   1:L PR[91] R[100]mm/sec CNT100;
   1:  PR[91,1] = PR[90,1] + 58.118;
   1:  PR[91,2] = PR[90,2] + -22.323;
   1:  PR[91,3] = PR[90,3] + 45.021;
   1:L PR[91] R[100]mm/sec CNT100;
   1:  PR[91,1] = PR[90,1] + 59.291;
   1:  PR[91,2] = PR[90,2] + -22.455;
   1:  PR[91,3] = PR[90,3] + 45.028;
   1:L PR[91] R[100]mm/sec CNT100;
   1:  PR[91,1] = PR[90,1] + 63.095;
   1:  PR[91,2] = PR[90,2] + -22.522;
   1:  PR[91,3] = PR[90,3] + 45.032;
   1:L PR[91] R[100]mm/sec CNT100;
   1:  PR[91,1] = PR[90,1] + 66.999;
   1:  PR[91,2] = PR[90,2] + -22.167;
   1:  PR[91,3] = PR[90,3] + 45.043;
   1:L PR[91] R[100]mm/sec CNT100;
   1:  PR[91,1] = PR[90,1] + 68.277;
   1:  PR[91,2] = PR[90,2] + -21.945;
   1:  PR[91,3] = PR[90,3] + 45.054;
   1:L PR[91] R[100]mm/sec CNT100;
   1:  PR[91,1] = PR[90,1] + 73.428;
   1:  PR[91,2] = PR[90,2] + -20.409;
   1:  PR[91,3] = PR[90,3] + 45.058;
   1:L PR[91] R[100]mm/sec CNT100;
   1:  PR[91,1] = PR[90,1] + 73.641;
   1:  PR[91,2] = PR[90,2] + -20.327;
   1:  PR[91,3] = PR[90,3] + 45.073;
   1:L PR[91] R[100]mm/sec CNT100;
   1:  PR[91,1] = PR[90,1] + 77.548;
   1:  PR[91,2] = PR[90,2] + -18.168;
   1:  PR[91,3] = PR[90,3] + 45.074;
   1:L PR[91] R[100]mm/sec CNT100;
   1:  PR[91,1] = PR[90,1] + 78.651;
   1:  PR[91,2] = PR[90,2] + -17.462;
   1:  PR[91,3] = PR[90,3] + 45.087;
   1:L PR[91] R[100]mm/sec CNT100;
   1:  PR[91,1] = PR[90,1] + 81.067;
   1:  PR[91,2] = PR[90,2] + -15.304;
   1:  PR[91,3] = PR[90,3] + 45.091;
   1:L PR[91] R[100]mm/sec CNT100;
   1:  PR[91,1] = PR[90,1] + 82.534;
   1:  PR[91,2] = PR[90,2] + -13.852;
   1:  PR[91,3] = PR[90,3] + 45.100;
   1:L PR[91] R[100]mm/sec CNT100;
   1:  PR[91,1] = PR[90,1] + 83.900;
   1:  PR[91,2] = PR[90,2] + -11.894;
   1:  PR[91,3] = PR[90,3] + 45.106;
   1:L PR[91] R[100]mm/sec CNT100;
   1:  PR[91,1] = PR[90,1] + 85.291;
   1:  PR[91,2] = PR[90,2] + -9.736;
   1:  PR[91,3] = PR[90,3] + 45.113;
   1:L PR[91] R[100]mm/sec CNT100;
   1:  PR[91,1] = PR[90,1] + 85.955;
   1:  PR[91,2] = PR[90,2] + -8.019;
   1:  PR[91,3] = PR[90,3] + 45.121;
   1:L PR[91] R[100]mm/sec CNT100;
   1:  PR[91,1] = PR[90,1] + 86.933;
   1:  PR[91,2] = PR[90,2] + -5.315;
   1:  PR[91,3] = PR[90,3] + 45.126;
   1:L PR[91] R[100]mm/sec CNT100;
   1:  PR[91,1] = PR[90,1] + 87.308;
   1:  PR[91,2] = PR[90,2] + -2.135;
   1:  PR[91,3] = PR[90,3] + 45.134;
   1:L PR[91] R[100]mm/sec CNT100;
   1:  PR[91,1] = PR[90,1] + 87.416;
   1:  PR[91,2] = PR[90,2] + -1.644;
   1:  PR[91,3] = PR[90,3] + 45.144;
   1:L PR[91] R[100]mm/sec CNT100;
   1:  PR[91,1] = PR[90,1] + 87.528;
   1:  PR[91,2] = PR[90,2] + -0.738;
   1:  PR[91,3] = PR[90,3] + 45.145;
   1:L PR[91] R[100]mm/sec CNT100;
   1:  PR[91,1] = PR[90,1] + 87.126;
   1:  PR[91,2] = PR[90,2] + 2.303;
   1:  PR[91,3] = PR[90,3] + 45.148;
   1:L PR[91] R[100]mm/sec CNT100;
   1:  PR[91,1] = PR[90,1] + 86.935;
   1:  PR[91,2] = PR[90,2] + 3.851;
   1:  PR[91,3] = PR[90,3] + 45.157;
   1:L PR[91] R[100]mm/sec CNT100;
   1:  PR[91,1] = PR[90,1] + 85.955;
   1:  PR[91,2] = PR[90,2] + 6.560;
   1:  PR[91,3] = PR[90,3] + 45.161;
   1:L PR[91] R[100]mm/sec CNT100;
   1:  PR[91,1] = PR[90,1] + 85.291;
   1:  PR[91,2] = PR[90,2] + 8.277;
   1:  PR[91,3] = PR[90,3] + 45.169;
   1:L PR[91] R[100]mm/sec CNT100;
   1:  PR[91,1] = PR[90,1] + 83.900;
   1:  PR[91,2] = PR[90,2] + 10.435;
   1:  PR[91,3] = PR[90,3] + 45.175;
   1:L PR[91] R[100]mm/sec CNT100;
   1:  PR[91,1] = PR[90,1] + 82.534;
   1:  PR[91,2] = PR[90,2] + 12.393;
   1:  PR[91,3] = PR[90,3] + 45.182;
   1:L PR[91] R[100]mm/sec CNT100;
   1:  PR[91,1] = PR[90,1] + 81.067;
   1:  PR[91,2] = PR[90,2] + 13.845;
   1:  PR[91,3] = PR[90,3] + 45.189;
   1:L PR[91] R[100]mm/sec CNT100;
   1:  PR[91,1] = PR[90,1] + 78.651;
   1:  PR[91,2] = PR[90,2] + 16.003;
   1:  PR[91,3] = PR[90,3] + 45.195;
   1:L PR[91] R[100]mm/sec CNT100;
   1:  PR[91,1] = PR[90,1] + 77.549;
   1:  PR[91,2] = PR[90,2] + 16.709;
   1:  PR[91,3] = PR[90,3] + 45.205;
   1:L PR[91] R[100]mm/sec CNT100;
   1:  PR[91,1] = PR[90,1] + 73.642;
   1:  PR[91,2] = PR[90,2] + 18.868;
   1:  PR[91,3] = PR[90,3] + 45.208;
   1:L PR[91] R[100]mm/sec CNT100;
   1:  PR[91,1] = PR[90,1] + 73.428;
   1:  PR[91,2] = PR[90,2] + 18.950;
   1:  PR[91,3] = PR[90,3] + 45.221;
   1:L PR[91] R[100]mm/sec CNT100;
   1:  PR[91,1] = PR[90,1] + 68.270;
   1:  PR[91,2] = PR[90,2] + 20.489;
   1:  PR[91,3] = PR[90,3] + 45.222;
   1:L PR[91] R[100]mm/sec CNT100;
   1:  PR[91,1] = PR[90,1] + 66.977;
   1:  PR[91,2] = PR[90,2] + 20.710;
   1:  PR[91,3] = PR[90,3] + 45.238;
   1:L PR[91] R[100]mm/sec CNT100;
   1:  PR[91,1] = PR[90,1] + 63.068;
   1:  PR[91,2] = PR[90,2] + 21.066;
   1:  PR[91,3] = PR[90,3] + 45.241;
   1:L PR[91] R[100]mm/sec CNT100;
   1:  PR[91,1] = PR[90,1] + 59.214;
   1:  PR[91,2] = PR[90,2] + 20.989;
   1:  PR[91,3] = PR[90,3] + 45.253;
   1:L PR[91] R[100]mm/sec CNT100;
   1:  PR[91,1] = PR[90,1] + 58.065;
   1:  PR[91,2] = PR[90,2] + 20.860;
   1:  PR[91,3] = PR[90,3] + 45.264;
   1:L PR[91] R[100]mm/sec CNT100;
   1:  PR[91,1] = PR[90,1] + 55.759;
   1:  PR[91,2] = PR[90,2] + 20.363;
   1:  PR[91,3] = PR[90,3] + 45.267;
   1:L PR[91] R[100]mm/sec CNT100;
   1:  PR[91,1] = PR[90,1] + 53.207;
   1:  PR[91,2] = PR[90,2] + 19.893;
   1:  PR[91,3] = PR[90,3] + 45.274;
   1:L PR[91] R[100]mm/sec CNT100;
   1:  PR[91,1] = PR[90,1] + 51.984;
   1:  PR[91,2] = PR[90,2] + 19.647;
   1:  PR[91,3] = PR[90,3] + 45.282;
   1:L PR[91] R[100]mm/sec CNT100;
   1:  PR[91,1] = PR[90,1] + 49.065;
   1:  PR[91,2] = PR[90,2] + 18.507;
   1:  PR[91,3] = PR[90,3] + 45.285;
   1:L PR[91] R[100]mm/sec CNT100;
   1:  PR[91,1] = PR[90,1] + 45.352;
   1:  PR[91,2] = PR[90,2] + 16.958;
   1:  PR[91,3] = PR[90,3] + 45.294;
   1:L PR[91] R[100]mm/sec CNT100;
   1:  PR[91,1] = PR[90,1] + 44.475;
   1:  PR[91,2] = PR[90,2] + 16.351;
   1:  PR[91,3] = PR[90,3] + 45.306;
   1:L PR[91] R[100]mm/sec CNT100;
   1:  PR[91,1] = PR[90,1] + 39.433;
   1:  PR[91,2] = PR[90,2] + 13.177;
   1:  PR[91,3] = PR[90,3] + 45.309;
   1:L PR[91] R[100]mm/sec CNT100;
   1:  PR[91,1] = PR[90,1] + 37.041;
   1:  PR[91,2] = PR[90,2] + 15.548;
   1:  PR[91,3] = PR[90,3] + 45.327;
   1:L PR[91] R[100]mm/sec CNT100;
   1:  PR[91,1] = PR[90,1] + 35.593;
   1:  PR[91,2] = PR[90,2] + 16.643;
   1:  PR[91,3] = PR[90,3] + 45.336;
   1:L PR[91] R[100]mm/sec CNT100;
   1:  PR[91,1] = PR[90,1] + 34.665;
   1:  PR[91,2] = PR[90,2] + 17.312;
   1:  PR[91,3] = PR[90,3] + 45.342;
   1:L PR[91] R[100]mm/sec CNT100;
   1:  PR[91,1] = PR[90,1] + 34.298;
   1:  PR[91,2] = PR[90,2] + 17.553;
   1:  PR[91,3] = PR[90,3] + 45.345;
   1:L PR[91] R[100]mm/sec CNT100;
   1:  PR[91,1] = PR[90,1] + 31.694;
   1:  PR[91,2] = PR[90,2] + 18.777;
   1:  PR[91,3] = PR[90,3] + 45.346;
   1:L PR[91] R[100]mm/sec CNT100;
   1:  PR[91,1] = PR[90,1] + 29.317;
   1:  PR[91,2] = PR[90,2] + 19.751;
   1:  PR[91,3] = PR[90,3] + 45.355;
   1:L PR[91] R[100]mm/sec CNT100;
   1:  PR[91,1] = PR[90,1] + 26.382;
   1:  PR[91,2] = PR[90,2] + 20.320;
   1:  PR[91,3] = PR[90,3] + 45.362;
   1:L PR[91] R[100]mm/sec CNT100;
   1:  PR[91,1] = PR[90,1] + 24.007;
   1:  PR[91,2] = PR[90,2] + 20.632;
   1:  PR[91,3] = PR[90,3] + 45.371;
   1:L PR[91] R[100]mm/sec CNT100;
   1:  PR[91,1] = PR[90,1] + 20.837;
   1:  PR[91,2] = PR[90,2] + 20.451;
   1:  PR[91,3] = PR[90,3] + 45.378;
   1:L PR[91] R[100]mm/sec CNT100;
   1:  PR[91,1] = PR[90,1] + 18.643;
   1:  PR[91,2] = PR[90,2] + 20.167;
   1:  PR[91,3] = PR[90,3] + 45.387;
   1:L PR[91] R[100]mm/sec CNT100;
   1:  PR[91,1] = PR[90,1] + 15.437;
   1:  PR[91,2] = PR[90,2] + 19.153;
   1:  PR[91,3] = PR[90,3] + 45.393;
   1:L PR[91] R[100]mm/sec CNT100;
   1:  PR[91,1] = PR[90,1] + 13.560;
   1:  PR[91,2] = PR[90,2] + 18.384;
   1:  PR[91,3] = PR[90,3] + 45.403;
   1:L PR[91] R[100]mm/sec CNT100;
   1:  PR[91,1] = PR[90,1] + 10.558;
   1:  PR[91,2] = PR[90,2] + 16.515;
   1:  PR[91,3] = PR[90,3] + 45.409;
   1:L PR[91] R[100]mm/sec CNT100;
   1:  PR[91,1] = PR[90,1] + 9.078;
   1:  PR[91,2] = PR[90,2] + 15.390;
   1:  PR[91,3] = PR[90,3] + 45.419;
   1:L PR[91] R[100]mm/sec CNT100;
   1:  PR[91,1] = PR[90,1] + 6.497;
   1:  PR[91,2] = PR[90,2] + 12.675;
   1:  PR[91,3] = PR[90,3] + 45.425;
   1:L PR[91] R[100]mm/sec CNT100;
   1:  PR[91,1] = PR[90,1] + 5.421;
   1:  PR[91,2] = PR[90,2] + 11.285;
   1:  PR[91,3] = PR[90,3] + 45.435;
   1:L PR[91] R[100]mm/sec CNT100;
   1:  PR[91,1] = PR[90,1] + 5.280;
   1:  PR[91,2] = PR[90,2] + 11.075;
   1:  PR[91,3] = PR[90,3] + 45.441;
   1:L PR[91] R[100]mm/sec CNT100;
   1:  PR[91,1] = PR[90,1] + 5.067;
   1:  PR[91,2] = PR[90,2] + 10.734;
   1:L PR[91] R[100]mm/sec CNT100;
   1:  PR[91,1] = PR[90,1] + 2.658;
   1:  PR[91,2] = PR[90,2] + 6.129;
   1:  PR[91,3] = PR[90,3] + 45.442;
   1:L PR[91] R[100]mm/sec CNT100;
   1:  PR[91,1] = PR[90,1] + 0.301;
   1:  PR[91,2] = PR[90,2] + 10.494;
   1:  PR[91,3] = PR[90,3] + 45.457;
   1:L PR[91] R[100]mm/sec CNT100;
   1:  PR[91,1] = PR[90,1] + -0.405;
   1:  PR[91,2] = PR[90,2] + 11.362;
   1:  PR[91,3] = PR[90,3] + 45.472;
   1:L PR[91] R[100]mm/sec CNT100;
   1:  PR[91,1] = PR[90,1] + -2.903;
   1:  PR[91,2] = PR[90,2] + 14.051;
   1:  PR[91,3] = PR[90,3] + 45.475;
   1:L PR[91] R[100]mm/sec CNT100;
   1:  PR[91,1] = PR[90,1] + -4.419;
   1:  PR[91,2] = PR[90,2] + 15.218;
   1:  PR[91,3] = PR[90,3] + 45.486;
   1:L PR[91] R[100]mm/sec CNT100;
   1:  PR[91,1] = PR[90,1] + -6.800;
   1:  PR[91,2] = PR[90,2] + 16.795;
   1:  PR[91,3] = PR[90,3] + 45.491;
   1:L PR[91] R[100]mm/sec CNT100;
   1:  PR[91,1] = PR[90,1] + -9.296;
   1:  PR[91,2] = PR[90,2] + 17.953;
   1:  PR[91,3] = PR[90,3] + 45.500;
   1:L PR[91] R[100]mm/sec CNT100;
   1:  PR[91,1] = PR[90,1] + -11.158;
   1:  PR[91,2] = PR[90,2] + 18.656;
   1:  PR[91,3] = PR[90,3] + 45.508;
   1:L PR[91] R[100]mm/sec CNT100;
   1:  PR[91,1] = PR[90,1] + -14.668;
   1:  PR[91,2] = PR[90,2] + 19.438;
   1:  PR[91,3] = PR[90,3] + 45.513;
   1:L PR[91] R[100]mm/sec CNT100;
   1:  PR[91,1] = PR[90,1] + -15.765;
   1:  PR[91,2] = PR[90,2] + 19.597;
   1:  PR[91,3] = PR[90,3] + 45.524;
   1:L PR[91] R[100]mm/sec CNT100;
   1:  PR[91,1] = PR[90,1] + -20.138;
   1:  PR[91,2] = PR[90,2] + 19.641;
   1:  PR[91,3] = PR[90,3] + 45.527;
   1:L PR[91] R[100]mm/sec CNT100;
   1:  PR[91,1] = PR[90,1] + -20.417;
   1:  PR[91,2] = PR[90,2] + 19.622;
   1:  PR[91,3] = PR[90,3] + 45.540;
   1:L PR[91] R[100]mm/sec CNT100;
   1:  PR[91,1] = PR[90,1] + -25.039;
   1:  PR[91,2] = PR[90,2] + 18.709;
   1:  PR[91,3] = PR[90,3] + 45.541;
   1:L PR[91] R[100]mm/sec CNT100;
   1:  PR[91,1] = PR[90,1] + -29.184;
   1:  PR[91,2] = PR[90,2] + 16.938;
   1:  PR[91,3] = PR[90,3] + 45.554;
   1:L PR[91] R[100]mm/sec CNT100;
   1:  PR[91,1] = PR[90,1] + -29.594;
   1:  PR[91,2] = PR[90,2] + 16.676;
   1:  PR[91,3] = PR[90,3] + 45.567;
   1:L PR[91] R[100]mm/sec CNT100;
   1:  PR[91,1] = PR[90,1] + -32.833;
   1:  PR[91,2] = PR[90,2] + 14.369;
   1:  PR[91,3] = PR[90,3] + 45.569;
   1:L PR[91] R[100]mm/sec CNT100;
   1:  PR[91,1] = PR[90,1] + -33.458;
   1:  PR[91,2] = PR[90,2] + 13.742;
   1:  PR[91,3] = PR[90,3] + 45.580;
   1:L PR[91] R[100]mm/sec CNT100;
   1:  PR[91,1] = PR[90,1] + -35.840;
   1:  PR[91,2] = PR[90,2] + 11.109;
   1:  PR[91,3] = PR[90,3] + 45.583;
   1:L PR[91] R[100]mm/sec CNT100;
   1:  PR[91,1] = PR[90,1] + -36.555;
   1:  PR[91,2] = PR[90,2] + 9.975;
   1:  PR[91,3] = PR[90,3] + 45.593;
   1:L PR[91] R[100]mm/sec CNT100;
   1:  PR[91,1] = PR[90,1] + -36.941;
   1:  PR[91,2] = PR[90,2] + 9.506;
   1:  PR[91,3] = PR[90,3] + 45.597;
   1:L PR[91] R[100]mm/sec CNT100;
   1:  PR[91,1] = PR[90,1] + -37.589;
   1:  PR[91,2] = PR[90,2] + 8.519;
   1:  PR[91,3] = PR[90,3] + 45.599;
   1:L PR[91] R[100]mm/sec CNT100;
   1:  PR[91,1] = PR[90,1] + -38.983;
   1:  PR[91,2] = PR[90,2] + 5.816;
   1:  PR[91,3] = PR[90,3] + 45.602;
   1:L PR[91] R[100]mm/sec CNT100;
   1:  PR[91,1] = PR[90,1] + -43.442;
   1:  PR[91,2] = PR[90,2] + 11.098;
   1:  PR[91,3] = PR[90,3] + 45.611;
   1:L PR[91] R[100]mm/sec CNT100;
   1:  PR[91,1] = PR[90,1] + -43.553;
   1:  PR[91,2] = PR[90,2] + 11.183;
   1:  PR[91,3] = PR[90,3] + 45.631;
   1:L PR[91] R[100]mm/sec CNT100;
   1:  PR[91,1] = PR[90,1] + -46.739;
   1:  PR[91,2] = PR[90,2] + 13.877;
   1:L PR[91] R[100]mm/sec CNT100;
   1:  PR[91,1] = PR[90,1] + -47.890;
   1:  PR[91,2] = PR[90,2] + 14.767;
   1:  PR[91,3] = PR[90,3] + 45.644;
   1:L PR[91] R[100]mm/sec CNT100;
   1:  PR[91,1] = PR[90,1] + -50.070;
   1:  PR[91,2] = PR[90,2] + 15.923;
   1:  PR[91,3] = PR[90,3] + 45.648;
   1:L PR[91] R[100]mm/sec CNT100;
   1:  PR[91,1] = PR[90,1] + -53.084;
   1:  PR[91,2] = PR[90,2] + 17.397;
   1:  PR[91,3] = PR[90,3] + 45.655;
   1:L PR[91] R[100]mm/sec CNT100;
   1:  PR[91,1] = PR[90,1] + -53.672;
   1:  PR[91,2] = PR[90,2] + 17.576;
   1:  PR[91,3] = PR[90,3] + 45.665;
   1:L PR[91] R[100]mm/sec CNT100;
   1:  PR[91,1] = PR[90,1] + -55.476;
   1:  PR[91,2] = PR[90,2] + 18.075;
   1:  PR[91,3] = PR[90,3] + 45.666;
   1:L PR[91] R[100]mm/sec CNT100;
   1:  PR[91,1] = PR[90,1] + -58.281;
   1:  PR[91,2] = PR[90,2] + 18.953;
   1:  PR[91,3] = PR[90,3] + 45.672;
   1:L PR[91] R[100]mm/sec CNT100;
   1:  PR[91,1] = PR[90,1] + -63.257;
   1:  PR[91,2] = PR[90,2] + 19.550;
   1:  PR[91,3] = PR[90,3] + 45.680;
   1:L PR[91] R[100]mm/sec CNT100;
   1:  PR[91] = PR[90];
   1:  PR[91,1] = PR[90,1] + -64.724;
   1:  PR[91,2] = PR[90,2] + 19.586;
   1:  PR[91,3] = PR[90,3] + 46.995;
   1:L PR[91] R[100]mm/sec CNT100;
   1:  PR[91,1] = PR[90,1] + -67.490;
   1:  PR[91,2] = PR[90,2] + 19.409;
   1:  PR[91,3] = PR[90,3] + 45.701;
   1:L PR[91] R[100]mm/sec CNT100;
   1:  PR[91,1] = PR[90,1] + -72.221;
   1:  PR[91,2] = PR[90,2] + 18.266;
   1:  PR[91,3] = PR[90,3] + 45.710;
   1:L PR[91] R[100]mm/sec CNT100;
   1:  PR[91,1] = PR[90,1] + -74.935;
   1:  PR[91,2] = PR[90,2] + 17.057;
   1:  PR[91,3] = PR[90,3] + 45.724;
   1:L PR[91] R[100]mm/sec CNT100;
   1:  PR[91,1] = PR[90,1] + -76.414;
   1:  PR[91,2] = PR[90,2] + 16.378;
   1:  PR[91,3] = PR[90,3] + 45.733;
   1:L PR[91] R[100]mm/sec CNT100;
   1:  PR[91,1] = PR[90,1] + -79.951;
   1:  PR[91,2] = PR[90,2] + 13.822;
   1:  PR[91,3] = PR[90,3] + 45.738;
   1:L PR[91] R[100]mm/sec CNT100;
   1:  PR[91,1] = PR[90,1] + -82.831;
   1:  PR[91,2] = PR[90,2] + 10.697;
   1:  PR[91,3] = PR[90,3] + 45.751;
   1:L PR[91] R[100]mm/sec CNT100;
   1:  PR[91,1] = PR[90,1] + -84.958;
   1:  PR[91,2] = PR[90,2] + 7.135;
   1:  PR[91,3] = PR[90,3] + 45.763;
   1:L PR[91] R[100]mm/sec CNT100;
   1:  PR[91,1] = PR[90,1] + -86.260;
   1:  PR[91,2] = PR[90,2] + 3.276;
   1:  PR[91,3] = PR[90,3] + 45.775;
   1:L PR[91] R[100]mm/sec CNT100;
   1:  PR[91,1] = PR[90,1] + -86.482;
   1:  PR[91,2] = PR[90,2] + 1.270;
   1:  PR[91,3] = PR[90,3] + 45.787;
   1:L PR[91] R[100]mm/sec CNT100;
   1:  PR[91,1] = PR[90,1] + -86.707;
   1:  PR[91,2] = PR[90,2] + 0.105;
   1:  PR[91,3] = PR[90,3] + 45.793;
   1:L PR[91] R[100]mm/sec CNT100;
   1:  PR[91,1] = PR[90,1] + -86.798;
   1:  PR[91,2] = PR[90,2] + -0.728;
   1:  PR[91,3] = PR[90,3] + 45.797;
   1:L PR[91] R[100]mm/sec CNT100;
   1:  PR[91,1] = PR[90,1] + -86.472;
   1:  PR[91,2] = PR[90,2] + -3.657;
   1:  PR[91,3] = PR[90,3] + 45.799;
   1:L PR[91] R[100]mm/sec CNT100;
   1:  PR[91,1] = PR[90,1] + -86.375;
   1:  PR[91,2] = PR[90,2] + -4.105;
   1:  PR[91,3] = PR[90,3] + 45.808;
   1:L PR[91] R[100]mm/sec CNT100;
   1:  PR[91,1] = PR[90,1] + -86.306;
   1:  PR[91,2] = PR[90,2] + -4.728;
   1:  PR[91,3] = PR[90,3] + 45.809;
   1:L PR[91] R[100]mm/sec CNT100;
   1:  PR[91,1] = PR[90,1] + -85.212;
   1:  PR[91,2] = PR[90,2] + -7.911;
   1:  PR[91,3] = PR[90,3] + 45.811;
   1:L PR[91] R[100]mm/sec CNT100;
   1:  PR[91,1] = PR[90,1] + -84.984;
   1:  PR[91,2] = PR[90,2] + -8.584;
   1:  PR[91,3] = PR[90,3] + 45.821;
   1:L PR[91] R[100]mm/sec CNT100;
   1:  PR[91,1] = PR[90,1] + -82.825;
   1:  PR[91,2] = PR[90,2] + -12.142;
   1:  PR[91,3] = PR[90,3] + 45.823;
   1:L PR[91] R[100]mm/sec CNT100;
   1:  PR[91,1] = PR[90,1] + -80.899;
   1:  PR[91,2] = PR[90,2] + -14.187;
   1:  PR[91,3] = PR[90,3] + 45.835;
   1:L PR[91] R[100]mm/sec CNT100;
   1:  PR[91,1] = PR[90,1] + -79.891;
   1:  PR[91,2] = PR[90,2] + -15.278;
   1:  PR[91,3] = PR[90,3] + 45.844;
   1:L PR[91] R[100]mm/sec CNT100;
   1:  PR[91,1] = PR[90,1] + -77.974;
   1:  PR[91,2] = PR[90,2] + -16.627;
   1:  PR[91,3] = PR[90,3] + 45.848;
   1:L PR[91] R[100]mm/sec CNT100;
   1:  PR[91,1] = PR[90,1] + -76.286;
   1:  PR[91,2] = PR[90,2] + -17.846;
   1:  PR[91,3] = PR[90,3] + 45.855;
   1:L PR[91] R[100]mm/sec CNT100;
   1:  PR[91,1] = PR[90,1] + -74.694;
   1:  PR[91,2] = PR[90,2] + -18.555;
   1:  PR[91,3] = PR[90,3] + 45.861;
   1:L PR[91] R[100]mm/sec CNT100;
   1:  PR[91,1] = PR[90,1] + -72.138;
   1:  PR[91,2] = PR[90,2] + -19.736;
   1:  PR[91,3] = PR[90,3] + 45.866;
   1:L PR[91] R[100]mm/sec CNT100;
   1:  PR[91,1] = PR[90,1] + -71.173;
   1:  PR[91,2] = PR[90,2] + -19.960;
   1:  PR[91,3] = PR[90,3] + 45.875;
   1:L PR[91] R[100]mm/sec CNT100;
   1:  PR[91,1] = PR[90,1] + -67.582;
   1:  PR[91,2] = PR[90,2] + -20.854;
   1:  PR[91,3] = PR[90,3] + 45.878;
   1:L PR[91] R[100]mm/sec CNT100;
   1:  PR[91,1] = PR[90,1] + -66.353;
   1:  PR[91,2] = PR[90,2] + -20.921;
   1:  PR[91,3] = PR[90,3] + 45.889;
   1:L PR[91] R[100]mm/sec CNT100;
   1:  PR[91,1] = PR[90,1] + -62.991;
   1:  PR[91,2] = PR[90,2] + -21.145;
   1:  PR[91,3] = PR[90,3] + 45.892;
   1:L PR[91] R[100]mm/sec CNT100;
   1:  PR[91,1] = PR[90,1] + -61.974;
   1:  PR[91,2] = PR[90,2] + -21.137;
   1:  PR[91,3] = PR[90,3] + 45.902;
   1:L PR[91] R[100]mm/sec CNT100;
   1:  PR[91,1] = PR[90,1] + -58.535;
   1:  PR[91,2] = PR[90,2] + -20.765;
   1:  PR[91,3] = PR[90,3] + 45.905;
   1:L PR[91] R[100]mm/sec CNT100;
   1:  PR[91,1] = PR[90,1] + -55.621;
   1:  PR[91,2] = PR[90,2] + -20.187;
   1:  PR[91,3] = PR[90,3] + 45.915;
   1:L PR[91] R[100]mm/sec CNT100;
   1:  PR[91,1] = PR[90,1] + -54.071;
   1:  PR[91,2] = PR[90,2] + -19.728;
   1:  PR[91,3] = PR[90,3] + 45.924;
   1:L PR[91] R[100]mm/sec CNT100;
   1:  PR[91,1] = PR[90,1] + -49.966;
   1:  PR[91,2] = PR[90,2] + -18.029;
   1:  PR[91,3] = PR[90,3] + 45.929;
   1:L PR[91] R[100]mm/sec CNT100;
   1:  PR[91,1] = PR[90,1] + -49.394;
   1:  PR[91,2] = PR[90,2] + -17.827;
   1:  PR[91,3] = PR[90,3] + 45.942;
   1:L PR[91] R[100]mm/sec CNT100;
   1:  PR[91,1] = PR[90,1] + -44.437;
   1:  PR[91,2] = PR[90,2] + -14.869;
   1:  PR[91,3] = PR[90,3] + 45.944;
   1:L PR[91] R[100]mm/sec CNT100;
   1:  PR[91,1] = PR[90,1] + -41.250;
   1:  PR[91,2] = PR[90,2] + -11.862;
   1:  PR[91,3] = PR[90,3] + 45.961;
   1:L PR[91] R[100]mm/sec CNT100;
   1:  PR[91,1] = PR[90,1] + -40.445;
   1:  PR[91,2] = PR[90,2] + -11.082;
   1:  PR[91,3] = PR[90,3] + 45.974;
   1:L PR[91] R[100]mm/sec CNT100;
   1:  PR[91,1] = PR[90,1] + -38.610;
   1:  PR[91,2] = PR[90,2] + -8.253;
   1:  PR[91,3] = PR[90,3] + 45.977;
   1:L PR[91] R[100]mm/sec CNT100;
   1:  PR[91,1] = PR[90,1] + -36.504;
   1:  PR[91,2] = PR[90,2] + -11.413;
   1:  PR[91,3] = PR[90,3] + 45.987;
   1:L PR[91] R[100]mm/sec CNT100;
   1:  PR[91,1] = PR[90,1] + -35.712;
   1:  PR[91,2] = PR[90,2] + -12.500;
   1:  PR[91,3] = PR[90,3] + 45.998;
   1:L PR[91] R[100]mm/sec CNT100;
   1:  PR[91,1] = PR[90,1] + -32.948;
   1:  PR[91,2] = PR[90,2] + -15.559;
   1:  PR[91,3] = PR[90,3] + 46.002;
   1:L PR[91] R[100]mm/sec CNT100;
   1:  PR[91,1] = PR[90,1] + -32.664;
   1:  PR[91,2] = PR[90,2] + -15.844;
   1:  PR[91,3] = PR[90,3] + 46.014;
   1:L PR[91] R[100]mm/sec CNT100;
   1:  PR[91,1] = PR[90,1] + -28.969;
   1:  PR[91,2] = PR[90,2] + -18.467;
   1:  PR[91,3] = PR[90,3] + 46.016;
   1:L PR[91] R[100]mm/sec CNT100;
   1:  PR[91,1] = PR[90,1] + -24.718;
   1:  PR[91,2] = PR[90,2] + -20.290;
   1:  PR[91,3] = PR[90,3] + 46.029;
   1:L PR[91] R[100]mm/sec CNT100;
   1:  PR[91,1] = PR[90,1] + -24.535;
   1:  PR[91,2] = PR[90,2] + -20.342;
   1:  PR[91,3] = PR[90,3] + 46.043;
   1:L PR[91] R[100]mm/sec CNT100;
   1:  PR[91,1] = PR[90,1] + -20.191;
   1:  PR[91,2] = PR[90,2] + -21.215;
   1:L PR[91] R[100]mm/sec CNT100;
   1:  PR[91,1] = PR[90,1] + -19.235;
   1:  PR[91,2] = PR[90,2] + -21.282;
   1:  PR[91,3] = PR[90,3] + 46.056;
   1:L PR[91] R[100]mm/sec CNT100;
   1:  PR[91,1] = PR[90,1] + -15.504;
   1:  PR[91,2] = PR[90,2] + -21.247;
   1:  PR[91,3] = PR[90,3] + 46.059;
   1:L PR[91] R[100]mm/sec CNT100;
   1:  PR[91,1] = PR[90,1] + -13.689;
   1:  PR[91,2] = PR[90,2] + -20.987;
   1:  PR[91,3] = PR[90,3] + 46.070;
   1:L PR[91] R[100]mm/sec CNT100;
   1:  PR[91,1] = PR[90,1] + -10.844;
   1:  PR[91,2] = PR[90,2] + -20.355;
   1:  PR[91,3] = PR[90,3] + 46.076;
   1:L PR[91] R[100]mm/sec CNT100;
   1:  PR[91,1] = PR[90,1] + -8.264;
   1:  PR[91,2] = PR[90,2] + -19.385;
   1:  PR[91,3] = PR[90,3] + 46.084;
   1:L PR[91] R[100]mm/sec CNT100;
   1:  PR[91,1] = PR[90,1] + -6.417;
   1:  PR[91,2] = PR[90,2] + -18.529;
   1:  PR[91,3] = PR[90,3] + 46.092;
   1:L PR[91] R[100]mm/sec CNT100;
   1:  PR[91,1] = PR[90,1] + -3.369;
   1:  PR[91,2] = PR[90,2] + -16.516;
   1:  PR[91,3] = PR[90,3] + 46.098;
   1:L PR[91] R[100]mm/sec CNT100;
   1:  PR[91,1] = PR[90,1] + -2.442;
   1:  PR[91,2] = PR[90,2] + -15.803;
   1:  PR[91,3] = PR[90,3] + 46.109;
   1:L PR[91] R[100]mm/sec CNT100;
   1:  PR[91,1] = PR[90,1] + 0.613;
   1:  PR[91,2] = PR[90,2] + -12.529;
   1:  PR[91,3] = PR[90,3] + 46.113;
   1:L PR[91] R[100]mm/sec CNT100;
   1:  PR[91,1] = PR[90,1] + 0.857;
   1:  PR[91,2] = PR[90,2] + -12.230;
   1:  PR[91,3] = PR[90,3] + 46.126;
   1:L PR[91] R[100]mm/sec CNT100;
   1:  PR[91,1] = PR[90,1] + 2.913;
   1:  PR[91,2] = PR[90,2] + -8.564;
   1:  PR[91,3] = PR[90,3] + 46.127;
   1:L PR[91] R[100]mm/sec CNT100;
   1:  PR[91,1] = PR[90,1] + 4.647;
   1:  PR[91,2] = PR[90,2] + -12.020;
   1:  PR[91,3] = PR[90,3] + 46.139;
   1:L PR[91] R[100]mm/sec CNT100;
   1:  PR[91,1] = PR[90,1] + 4.706;
   1:  PR[91,2] = PR[90,2] + -12.096;
   1:  PR[91,3] = PR[90,3] + 46.151;
   1:L PR[91] R[100]mm/sec CNT100;
   1:  PR[91,1] = PR[90,1] + 5.116;
   1:  PR[91,2] = PR[90,2] + -12.707;
   1:L PR[91] R[100]mm/sec CNT100;
   1:  PR[91,1] = PR[90,1] + 6.042;
   1:  PR[91,2] = PR[90,2] + -14.022;
   1:  PR[91,3] = PR[90,3] + 46.153;
   1:L PR[91] R[100]mm/sec CNT100;
   1:  PR[91,1] = PR[90,1] + 8.993;
   1:  PR[91,2] = PR[90,2] + -17.132;
   1:  PR[91,3] = PR[90,3] + 46.158;
   1:L PR[91] R[100]mm/sec CNT100;
   1:  PR[91,1] = PR[90,1] + 10.043;
   1:  PR[91,2] = PR[90,2] + -17.928;
   1:  PR[91,3] = PR[90,3] + 46.171;
   1:L PR[91] R[100]mm/sec CNT100;
   1:  PR[91,1] = PR[90,1] + 13.529;
   1:  PR[91,2] = PR[90,2] + -20.101;
   1:  PR[91,3] = PR[90,3] + 46.174;
   1:L PR[91] R[100]mm/sec CNT100;
   1:  PR[91,1] = PR[90,1] + 14.911;
   1:  PR[91,2] = PR[90,2] + -20.665;
   1:  PR[91,3] = PR[90,3] + 46.187;
   1:L PR[91] R[100]mm/sec CNT100;
   1:  PR[91,1] = PR[90,1] + 18.656;
   1:  PR[91,2] = PR[90,2] + -21.851;
   1:  PR[91,3] = PR[90,3] + 46.191;
   1:L PR[91] R[100]mm/sec CNT100;
   1:  PR[91,1] = PR[90,1] + 20.325;
   1:  PR[91,2] = PR[90,2] + -22.065;
   1:  PR[91,3] = PR[90,3] + 46.203;
   1:L PR[91] R[100]mm/sec CNT100;
   1:  PR[91,1] = PR[90,1] + 24.054;
   1:  PR[91,2] = PR[90,2] + -22.279;
   1:  PR[91,3] = PR[90,3] + 46.208;
   1:L PR[91] R[100]mm/sec CNT100;
   1:  PR[91,1] = PR[90,1] + 25.912;
   1:  PR[91,2] = PR[90,2] + -22.032;
   1:  PR[91,3] = PR[90,3] + 46.219;
   1:L PR[91] R[100]mm/sec CNT100;
   1:  PR[91,1] = PR[90,1] + 29.388;
   1:  PR[91,2] = PR[90,2] + -21.358;
   1:  PR[91,3] = PR[90,3] + 46.224;
   1:L PR[91] R[100]mm/sec CNT100;
   1:  PR[91,1] = PR[90,1] + 31.288;
   1:  PR[91,2] = PR[90,2] + -20.575;
   1:  PR[91,3] = PR[90,3] + 46.235;
   1:L PR[91] R[100]mm/sec CNT100;
   1:  PR[91,1] = PR[90,1] + 34.325;
   1:  PR[91,2] = PR[90,2] + -19.148;
   1:  PR[91,3] = PR[90,3] + 46.241;
   1:L PR[91] R[100]mm/sec CNT100;
   1:  PR[91,1] = PR[90,1] + 36.232;
   1:  PR[91,2] = PR[90,2] + -17.701;
   1:  PR[91,3] = PR[90,3] + 46.251;
   1:L PR[91] R[100]mm/sec CNT100;
   1:  PR[91,1] = PR[90,1] + 36.567;
   1:  PR[91,2] = PR[90,2] + -17.517;
   1:  PR[91,3] = PR[90,3] + 46.258;
   1:L PR[91] R[100]mm/sec CNT100;
   1:  PR[91,1] = PR[90,1] + 36.907;
   1:  PR[91,2] = PR[90,2] + -17.286;
   1:  PR[91,3] = PR[90,3] + 46.259;
   1:L PR[91] R[100]mm/sec CNT100;
   1:  PR[91,1] = PR[90,1] + 38.811;
   1:  PR[91,2] = PR[90,2] + -15.517;
   1:  PR[91,3] = PR[90,3] + 46.260;
   1:L PR[91] R[100]mm/sec CNT100;
   1:  PR[91,1] = PR[90,1] + 43.245;
   1:  PR[91,2] = PR[90,2] + -18.271;
   1:  PR[91,3] = PR[90,3] + 46.268;
   1:L PR[91] R[100]mm/sec CNT100;
   1:  PR[91,1] = PR[90,1] + 44.092;
   1:  PR[91,2] = PR[90,2] + -18.697;
   1:  PR[91,3] = PR[90,3] + 46.283;
   1:L PR[91] R[100]mm/sec CNT100;
   1:  PR[91,1] = PR[90,1] + 45.603;
   1:  PR[91,2] = PR[90,2] + -19.249;
   1:  PR[91,3] = PR[90,3] + 46.286;
   1:L PR[91] R[100]mm/sec CNT100;
   1:  PR[91,1] = PR[90,1] + 48.808;
   1:  PR[91,2] = PR[90,2] + -20.595;
   1:  PR[91,3] = PR[90,3] + 46.291;
   1:L PR[91] R[100]mm/sec CNT100;
   1:  PR[91,1] = PR[90,1] + 50.641;
   1:  PR[91,2] = PR[90,2] + -21.303;
   1:  PR[91,3] = PR[90,3] + 46.301;
   1:L PR[91] R[100]mm/sec CNT100;
   1:  PR[91,1] = PR[90,1] + 53.057;
   1:  PR[91,2] = PR[90,2] + -21.795;
   1:  PR[91,3] = PR[90,3] + 46.307;
   1:L PR[91] R[100]mm/sec CNT100;
   1:  PR[91,1] = PR[90,1] + 57.754;
   1:  PR[91,2] = PR[90,2] + -22.648;
   1:  PR[91,3] = PR[90,3] + 46.314;
   1:L PR[91] R[100]mm/sec CNT100;
   1:  PR[91,1] = PR[90,1] + 62.766;
   1:  PR[91,2] = PR[90,2] + -22.736;
   1:  PR[91,3] = PR[90,3] + 46.328;
   1:L PR[91] R[100]mm/sec CNT100;
   1:  PR[91,1] = PR[90,1] + 65.485;
   1:  PR[91,2] = PR[90,2] + -22.489;
   1:  PR[91,3] = PR[90,3] + 46.343;
   1:L PR[91] R[100]mm/sec CNT100;
   1:  PR[91,1] = PR[90,1] + 67.903;
   1:  PR[91,2] = PR[90,2] + -22.069;
   1:  PR[91,3] = PR[90,3] + 46.351;
   1:L PR[91] R[100]mm/sec CNT100;
   1:  PR[91,1] = PR[90,1] + 72.807;
   1:  PR[91,2] = PR[90,2] + -20.596;
   1:  PR[91,3] = PR[90,3] + 46.358;
   1:L PR[91] R[100]mm/sec CNT100;
   1:  PR[91,1] = PR[90,1] + 73.002;
   1:  PR[91,2] = PR[90,2] + -20.523;
   1:  PR[91,3] = PR[90,3] + 46.373;
   1:L PR[91] R[100]mm/sec CNT100;
   1:  PR[91,1] = PR[90,1] + 77.452;
   1:  PR[91,2] = PR[90,2] + -18.074;
   1:  PR[91,3] = PR[90,3] + 46.374;
   1:L PR[91] R[100]mm/sec CNT100;
   1:  PR[91,1] = PR[90,1] + 78.000;
   1:  PR[91,2] = PR[90,2] + -17.723;
   1:  PR[91,3] = PR[90,3] + 46.389;
   1:L PR[91] R[100]mm/sec CNT100;
   1:  PR[91,1] = PR[90,1] + 80.949;
   1:  PR[91,2] = PR[90,2] + -15.089;
   1:  PR[91,3] = PR[90,3] + 46.391;
   1:L PR[91] R[100]mm/sec CNT100;
   1:  PR[91,1] = PR[90,1] + 81.984;
   1:  PR[91,2] = PR[90,2] + -14.064;
   1:  PR[91,3] = PR[90,3] + 46.402;
   1:L PR[91] R[100]mm/sec CNT100;
   1:  PR[91,1] = PR[90,1] + 83.732;
   1:  PR[91,2] = PR[90,2] + -11.559;
   1:  PR[91,3] = PR[90,3] + 46.407;
   1:L PR[91] R[100]mm/sec CNT100;
   1:  PR[91,1] = PR[90,1] + 84.811;
   1:  PR[91,2] = PR[90,2] + -9.884;
   1:  PR[91,3] = PR[90,3] + 46.416;
   1:L PR[91] R[100]mm/sec CNT100;
   1:  PR[91,1] = PR[90,1] + 85.707;
   1:  PR[91,2] = PR[90,2] + -7.566;
   1:  PR[91,3] = PR[90,3] + 46.422;
   1:L PR[91] R[100]mm/sec CNT100;
   1:  PR[91,1] = PR[90,1] + 86.494;
   1:  PR[91,2] = PR[90,2] + -5.391;
   1:  PR[91,3] = PR[90,3] + 46.429;
   1:L PR[91] R[100]mm/sec CNT100;
   1:  PR[91,1] = PR[90,1] + 86.799;
   1:  PR[91,2] = PR[90,2] + -2.806;
   1:  PR[91,3] = PR[90,3] + 46.436;
   1:L PR[91] R[100]mm/sec CNT100;
   1:  PR[91,1] = PR[90,1] + 86.888;
   1:  PR[91,2] = PR[90,2] + -2.403;
   1:  PR[91,3] = PR[90,3] + 46.444;
   1:L PR[91] R[100]mm/sec CNT100;
   1:  PR[91,1] = PR[90,1] + 87.094;
   1:  PR[91,2] = PR[90,2] + -0.738;
   1:  PR[91,3] = PR[90,3] + 46.445;
   1:L PR[91] R[100]mm/sec CNT100;
   1:  PR[91,1] = PR[90,1] + 86.765;
   1:  PR[91,2] = PR[90,2] + 1.744;
   1:  PR[91,3] = PR[90,3] + 46.450;
   1:L PR[91] R[100]mm/sec CNT100;
   1:  PR[91,1] = PR[90,1] + 86.496;
   1:  PR[91,2] = PR[90,2] + 3.927;
   1:  PR[91,3] = PR[90,3] + 46.457;
   1:L PR[91] R[100]mm/sec CNT100;
   1:  PR[91,1] = PR[90,1] + 85.707;
   1:  PR[91,2] = PR[90,2] + 6.107;
   1:  PR[91,3] = PR[90,3] + 46.464;
   1:L PR[91] R[100]mm/sec CNT100;
   1:  PR[91,1] = PR[90,1] + 84.811;
   1:  PR[91,2] = PR[90,2] + 8.425;
   1:  PR[91,3] = PR[90,3] + 46.470;
   1:L PR[91] R[100]mm/sec CNT100;
   1:  PR[91,1] = PR[90,1] + 83.732;
   1:  PR[91,2] = PR[90,2] + 10.100;
   1:  PR[91,3] = PR[90,3] + 46.478;
   1:L PR[91] R[100]mm/sec CNT100;
   1:  PR[91,1] = PR[90,1] + 81.984;
   1:  PR[91,2] = PR[90,2] + 12.605;
   1:  PR[91,3] = PR[90,3] + 46.484;
   1:L PR[91] R[100]mm/sec CNT100;
   1:  PR[91,1] = PR[90,1] + 80.949;
   1:  PR[91,2] = PR[90,2] + 13.630;
   1:  PR[91,3] = PR[90,3] + 46.493;
   1:L PR[91] R[100]mm/sec CNT100;
   1:  PR[91,1] = PR[90,1] + 78.000;
   1:  PR[91,2] = PR[90,2] + 16.264;
   1:  PR[91,3] = PR[90,3] + 46.497;
   1:L PR[91] R[100]mm/sec CNT100;
   1:  PR[91,1] = PR[90,1] + 77.453;
   1:  PR[91,2] = PR[90,2] + 16.614;
   1:  PR[91,3] = PR[90,3] + 46.509;
   1:L PR[91] R[100]mm/sec CNT100;
   1:  PR[91,1] = PR[90,1] + 73.002;
   1:  PR[91,2] = PR[90,2] + 19.064;
   1:  PR[91,3] = PR[90,3] + 46.511;
   1:L PR[91] R[100]mm/sec CNT100;
   1:  PR[91,1] = PR[90,1] + 72.804;
   1:  PR[91,2] = PR[90,2] + 19.138;
   1:  PR[91,3] = PR[90,3] + 46.526;
   1:L PR[91] R[100]mm/sec CNT100;
   1:  PR[91,1] = PR[90,1] + 67.889;
   1:  PR[91,2] = PR[90,2] + 20.615;
   1:L PR[91] R[100]mm/sec CNT100;
   1:  PR[91,1] = PR[90,1] + 65.442;
   1:  PR[91,2] = PR[90,2] + 21.034;
   1:  PR[91,3] = PR[90,3] + 46.541;
   1:L PR[91] R[100]mm/sec CNT100;
   1:  PR[91,1] = PR[90,1] + 62.730;
   1:  PR[91,2] = PR[90,2] + 21.281;
   1:  PR[91,3] = PR[90,3] + 46.549;
   1:L PR[91] R[100]mm/sec CNT100;
   1:  PR[91,1] = PR[90,1] + 57.700;
   1:  PR[91,2] = PR[90,2] + 21.181;
   1:  PR[91,3] = PR[90,3] + 46.557;
   1:L PR[91] R[100]mm/sec CNT100;
   1:  PR[91,1] = PR[90,1] + 53.020;
   1:  PR[91,2] = PR[90,2] + 20.321;
   1:  PR[91,3] = PR[90,3] + 46.572;
   1:L PR[91] R[100]mm/sec CNT100;
   1:  PR[91,1] = PR[90,1] + 50.620;
   1:  PR[91,2] = PR[90,2] + 19.838;
   1:  PR[91,3] = PR[90,3] + 46.586;
   1:L PR[91] R[100]mm/sec CNT100;
   1:  PR[91,1] = PR[90,1] + 48.808;
   1:  PR[91,2] = PR[90,2] + 19.130;
   1:  PR[91,3] = PR[90,3] + 46.593;
   1:L PR[91] R[100]mm/sec CNT100;
   1:  PR[91,1] = PR[90,1] + 45.600;
   1:  PR[91,2] = PR[90,2] + 17.792;
   1:  PR[91,3] = PR[90,3] + 46.599;
   1:L PR[91] R[100]mm/sec CNT100;
   1:  PR[91,1] = PR[90,1] + 44.120;
   1:  PR[91,2] = PR[90,2] + 17.252;
   1:  PR[91,3] = PR[90,3] + 46.609;
   1:L PR[91] R[100]mm/sec CNT100;
   1:  PR[91,1] = PR[90,1] + 43.292;
   1:  PR[91,2] = PR[90,2] + 16.836;
   1:  PR[91,3] = PR[90,3] + 46.614;
   1:L PR[91] R[100]mm/sec CNT100;
   1:  PR[91,1] = PR[90,1] + 38.759;
   1:  PR[91,2] = PR[90,2] + 13.983;
   1:  PR[91,3] = PR[90,3] + 46.616;
   1:L PR[91] R[100]mm/sec CNT100;
   1:  PR[91,1] = PR[90,1] + 36.835;
   1:  PR[91,2] = PR[90,2] + 15.889;
   1:  PR[91,3] = PR[90,3] + 46.632;
   1:L PR[91] R[100]mm/sec CNT100;
   1:  PR[91,1] = PR[90,1] + 35.929;
   1:  PR[91,2] = PR[90,2] + 16.574;
   1:  PR[91,3] = PR[90,3] + 46.640;
   1:L PR[91] R[100]mm/sec CNT100;
   1:  PR[91,1] = PR[90,1] + 34.828;
   1:  PR[91,2] = PR[90,2] + 17.369;
   1:  PR[91,3] = PR[90,3] + 46.643;
   1:L PR[91] R[100]mm/sec CNT100;
   1:  PR[91,1] = PR[90,1] + 34.369;
   1:  PR[91,2] = PR[90,2] + 17.671;
   1:  PR[91,3] = PR[90,3] + 46.647;
   1:L PR[91] R[100]mm/sec CNT100;
   1:  PR[91,1] = PR[90,1] + 31.274;
   1:  PR[91,2] = PR[90,2] + 19.125;
   1:  PR[91,3] = PR[90,3] + 46.649;
   1:L PR[91] R[100]mm/sec CNT100;
   1:  PR[91,1] = PR[90,1] + 29.376;
   1:  PR[91,2] = PR[90,2] + 19.903;
   1:  PR[91,3] = PR[90,3] + 46.659;
   1:L PR[91] R[100]mm/sec CNT100;
   1:  PR[91,1] = PR[90,1] + 25.901;
   1:  PR[91,2] = PR[90,2] + 20.577;
   1:  PR[91,3] = PR[90,3] + 46.665;
   1:L PR[91] R[100]mm/sec CNT100;
   1:  PR[91,1] = PR[90,1] + 24.046;
   1:  PR[91,2] = PR[90,2] + 20.820;
   1:  PR[91,3] = PR[90,3] + 46.676;
   1:L PR[91] R[100]mm/sec CNT100;
   1:  PR[91,1] = PR[90,1] + 20.320;
   1:  PR[91,2] = PR[90,2] + 20.607;
   1:  PR[91,3] = PR[90,3] + 46.681;
   1:L PR[91] R[100]mm/sec CNT100;
   1:  PR[91,1] = PR[90,1] + 18.653;
   1:  PR[91,2] = PR[90,2] + 20.391;
   1:  PR[91,3] = PR[90,3] + 46.692;
   1:L PR[91] R[100]mm/sec CNT100;
   1:  PR[91,1] = PR[90,1] + 14.910;
   1:  PR[91,2] = PR[90,2] + 19.208;
   1:  PR[91,3] = PR[90,3] + 46.697;
   1:L PR[91] R[100]mm/sec CNT100;
   1:  PR[91,1] = PR[90,1] + 13.530;
   1:  PR[91,2] = PR[90,2] + 18.643;
   1:  PR[91,3] = PR[90,3] + 46.709;
   1:L PR[91] R[100]mm/sec CNT100;
   1:  PR[91,1] = PR[90,1] + 10.046;
   1:  PR[91,2] = PR[90,2] + 16.472;
   1:  PR[91,3] = PR[90,3] + 46.713;
   1:L PR[91] R[100]mm/sec CNT100;
   1:  PR[91,1] = PR[90,1] + 8.998;
   1:  PR[91,2] = PR[90,2] + 15.676;
   1:  PR[91,3] = PR[90,3] + 46.725;
   1:L PR[91] R[100]mm/sec CNT100;
   1:  PR[91,1] = PR[90,1] + 6.015;
   1:  PR[91,2] = PR[90,2] + 12.539;
   1:  PR[91,3] = PR[90,3] + 46.729;
   1:L PR[91] R[100]mm/sec CNT100;
   1:  PR[91,1] = PR[90,1] + 5.291;
   1:  PR[91,2] = PR[90,2] + 11.603;
   1:  PR[91,3] = PR[90,3] + 46.742;
   1:L PR[91] R[100]mm/sec CNT100;
   1:  PR[91,1] = PR[90,1] + 4.852;
   1:  PR[91,2] = PR[90,2] + 10.922;
   1:  PR[91,3] = PR[90,3] + 46.745;
   1:L PR[91] R[100]mm/sec CNT100;
   1:  PR[91,1] = PR[90,1] + 2.845;
   1:  PR[91,2] = PR[90,2] + 7.085;
   1:  PR[91,3] = PR[90,3] + 46.748;
   1:L PR[91] R[100]mm/sec CNT100;
   1:  PR[91,1] = PR[90,1] + 0.861;
   1:  PR[91,2] = PR[90,2] + 10.761;
   1:  PR[91,3] = PR[90,3] + 46.761;
   1:L PR[91] R[100]mm/sec CNT100;
   1:  PR[91,1] = PR[90,1] + 0.644;
   1:  PR[91,2] = PR[90,2] + 11.027;
   1:  PR[91,3] = PR[90,3] + 46.773;
   1:L PR[91] R[100]mm/sec CNT100;
   1:  PR[91,1] = PR[90,1] + -2.423;
   1:  PR[91,2] = PR[90,2] + 14.328;
   1:  PR[91,3] = PR[90,3] + 46.774;
   1:L PR[91] R[100]mm/sec CNT100;
   1:  PR[91,1] = PR[90,1] + -3.347;
   1:  PR[91,2] = PR[90,2] + 15.039;
   1:  PR[91,3] = PR[90,3] + 46.787;
   1:L PR[91] R[100]mm/sec CNT100;
   1:  PR[91,1] = PR[90,1] + -6.396;
   1:  PR[91,2] = PR[90,2] + 17.059;
   1:  PR[91,3] = PR[90,3] + 46.791;
   1:L PR[91] R[100]mm/sec CNT100;
   1:  PR[91,1] = PR[90,1] + -8.240;
   1:  PR[91,2] = PR[90,2] + 17.915;
   1:  PR[91,3] = PR[90,3] + 46.802;
   1:L PR[91] R[100]mm/sec CNT100;
   1:  PR[91,1] = PR[90,1] + -10.822;
   1:  PR[91,2] = PR[90,2] + 18.890;
   1:  PR[91,3] = PR[90,3] + 46.808;
   1:L PR[91] R[100]mm/sec CNT100;
   1:  PR[91,1] = PR[90,1] + -13.665;
   1:  PR[91,2] = PR[90,2] + 19.523;
   1:  PR[91,3] = PR[90,3] + 46.816;
   1:L PR[91] R[100]mm/sec CNT100;
   1:  PR[91,1] = PR[90,1] + -15.484;
   1:  PR[91,2] = PR[90,2] + 19.787;
   1:  PR[91,3] = PR[90,3] + 46.824;
   1:L PR[91] R[100]mm/sec CNT100;
   1:  PR[91,1] = PR[90,1] + -19.214;
   1:  PR[91,2] = PR[90,2] + 19.824;
   1:  PR[91,3] = PR[90,3] + 46.830;
   1:L PR[91] R[100]mm/sec CNT100;
   1:  PR[91,1] = PR[90,1] + -20.173;
   1:  PR[91,2] = PR[90,2] + 19.758;
   1:  PR[91,3] = PR[90,3] + 46.841;
   1:L PR[91] R[100]mm/sec CNT100;
   1:  PR[91,1] = PR[90,1] + -24.519;
   1:  PR[91,2] = PR[90,2] + 18.888;
   1:  PR[91,3] = PR[90,3] + 46.844;
   1:L PR[91] R[100]mm/sec CNT100;
   1:  PR[91,1] = PR[90,1] + -24.704;
   1:  PR[91,2] = PR[90,2] + 18.835;
   1:  PR[91,3] = PR[90,3] + 46.857;
   1:L PR[91] R[100]mm/sec CNT100;
   1:  PR[91,1] = PR[90,1] + -28.958;
   1:  PR[91,2] = PR[90,2] + 17.014;
   1:L PR[91] R[100]mm/sec CNT100;
   1:  PR[91,1] = PR[90,1] + -32.655;
   1:  PR[91,2] = PR[90,2] + 14.393;
   1:  PR[91,3] = PR[90,3] + 46.871;
   1:L PR[91] R[100]mm/sec CNT100;
   1:  PR[91,1] = PR[90,1] + -32.939;
   1:  PR[91,2] = PR[90,2] + 14.108;
   1:  PR[91,3] = PR[90,3] + 46.884;
   1:L PR[91] R[100]mm/sec CNT100;
   1:  PR[91,1] = PR[90,1] + -35.657;
   1:  PR[91,2] = PR[90,2] + 11.104;
   1:  PR[91,3] = PR[90,3] + 46.885;
   1:L PR[91] R[100]mm/sec CNT100;
   1:  PR[91,1] = PR[90,1] + -36.124;
   1:  PR[91,2] = PR[90,2] + 10.362;
   1:  PR[91,3] = PR[90,3] + 46.897;
   1:L PR[91] R[100]mm/sec CNT100;
   1:  PR[91,1] = PR[90,1] + -36.562;
   1:  PR[91,2] = PR[90,2] + 9.831;
   1:  PR[91,3] = PR[90,3] + 46.900;
   1:L PR[91] R[100]mm/sec CNT100;
   1:  PR[91,1] = PR[90,1] + -38.369;
   1:  PR[91,2] = PR[90,2] + 7.077;
   1:  PR[91,3] = PR[90,3] + 46.902;
   1:L PR[91] R[100]mm/sec CNT100;
   1:  PR[91,1] = PR[90,1] + -41.729;
   1:  PR[91,2] = PR[90,2] + 11.034;
   1:  PR[91,3] = PR[90,3] + 46.912;
   1:L PR[91] R[100]mm/sec CNT100;
   1:  PR[91,1] = PR[90,1] + -42.758;
   1:  PR[91,2] = PR[90,2] + 11.864;
   1:  PR[91,3] = PR[90,3] + 46.927;
   1:L PR[91] R[100]mm/sec CNT100;
   1:  PR[91,1] = PR[90,1] + -45.200;
   1:  PR[91,2] = PR[90,2] + 13.677;
   1:  PR[91,3] = PR[90,3] + 46.931;
   1:L PR[91] R[100]mm/sec CNT100;
   1:  PR[91,1] = PR[90,1] + -46.269;
   1:  PR[91,2] = PR[90,2] + 14.581;
   1:  PR[91,3] = PR[90,3] + 46.940;
   1:L PR[91] R[100]mm/sec CNT100;
   1:  PR[91,1] = PR[90,1] + -46.536;
   1:  PR[91,2] = PR[90,2] + 14.788;
   1:  PR[91,3] = PR[90,3] + 46.944;
   1:L PR[91] R[100]mm/sec CNT100;
   1:  PR[91,1] = PR[90,1] + -49.722;
   1:  PR[91,2] = PR[90,2] + 16.478;
   1:  PR[91,3] = PR[90,3] + 46.945;
   1:L PR[91] R[100]mm/sec CNT100;
   1:  PR[91,1] = PR[90,1] + -51.804;
   1:  PR[91,2] = PR[90,2] + 17.496;
   1:  PR[91,3] = PR[90,3] + 46.956;
   1:L PR[91] R[100]mm/sec CNT100;
   1:  PR[91,1] = PR[90,1] + -53.403;
   1:  PR[91,2] = PR[90,2] + 17.983;
   1:  PR[91,3] = PR[90,3] + 46.963;
   1:L PR[91] R[100]mm/sec CNT100;
   1:  PR[91,1] = PR[90,1] + -57.477;
   1:  PR[91,2] = PR[90,2] + 19.112;
   1:  PR[91,3] = PR[90,3] + 46.968;
   1:L PR[91] R[100]mm/sec CNT100;
   1:  PR[91,1] = PR[90,1] + -62.528;
   1:  PR[91,2] = PR[90,2] + 19.707;
   1:  PR[91,3] = PR[90,3] + 46.980;
   1:L PR[91] R[100]mm/sec CNT100;
   1:  PR[91] = PR[90];
   1:  PR[91,1] = PR[90,1] + -66.803;
   1:  PR[91,2] = PR[90,2] + 19.552;
   1:  PR[91,3] = PR[90,3] + 48.295;
   1:L PR[91] R[100]mm/sec CNT100;
   1:  PR[91,1] = PR[90,1] + -69.693;
   1:  PR[91,2] = PR[90,2] + 18.858;
   1:  PR[91,3] = PR[90,3] + 47.010;
   1:L PR[91] R[100]mm/sec CNT100;
   1:  PR[91,1] = PR[90,1] + -71.553;
   1:  PR[91,2] = PR[90,2] + 18.395;
   1:  PR[91,3] = PR[90,3] + 47.019;
   1:L PR[91] R[100]mm/sec CNT100;
   1:  PR[91,1] = PR[90,1] + -75.615;
   1:  PR[91,2] = PR[90,2] + 16.586;
   1:  PR[91,3] = PR[90,3] + 47.025;
   1:L PR[91] R[100]mm/sec CNT100;
   1:  PR[91,1] = PR[90,1] + -75.879;
   1:  PR[91,2] = PR[90,2] + 16.466;
   1:  PR[91,3] = PR[90,3] + 47.038;
   1:L PR[91] R[100]mm/sec CNT100;
   1:  PR[91,1] = PR[90,1] + -77.325;
   1:  PR[91,2] = PR[90,2] + 15.458;
   1:  PR[91,3] = PR[90,3] + 47.039;
   1:L PR[91] R[100]mm/sec CNT100;
   1:  PR[91,1] = PR[90,1] + -79.487;
   1:  PR[91,2] = PR[90,2] + 13.894;
   1:  PR[91,3] = PR[90,3] + 47.045;
   1:L PR[91] R[100]mm/sec CNT100;
   1:  PR[91,1] = PR[90,1] + -82.377;
   1:  PR[91,2] = PR[90,2] + 10.752;
   1:  PR[91,3] = PR[90,3] + 47.053;
   1:L PR[91] R[100]mm/sec CNT100;
   1:  PR[91,1] = PR[90,1] + -84.512;
   1:  PR[91,2] = PR[90,2] + 7.172;
   1:  PR[91,3] = PR[90,3] + 47.066;
   1:L PR[91] R[100]mm/sec CNT100;
   1:  PR[91,1] = PR[90,1] + -85.818;
   1:  PR[91,2] = PR[90,2] + 3.294;
   1:  PR[91,3] = PR[90,3] + 47.078;
   1:L PR[91] R[100]mm/sec CNT100;
   1:  PR[91,1] = PR[90,1] + -85.980;
   1:  PR[91,2] = PR[90,2] + 1.831;
   1:  PR[91,3] = PR[90,3] + 47.091;
   1:L PR[91] R[100]mm/sec CNT100;
   1:  PR[91,1] = PR[90,1] + -86.148;
   1:  PR[91,2] = PR[90,2] + 0.962;
   1:  PR[91,3] = PR[90,3] + 47.095;
   1:L PR[91] R[100]mm/sec CNT100;
   1:  PR[91,1] = PR[90,1] + -86.333;
   1:  PR[91,2] = PR[90,2] + -0.728;
   1:  PR[91,3] = PR[90,3] + 47.098;
   1:L PR[91] R[100]mm/sec CNT100;
   1:  PR[91,1] = PR[90,1] + -86.094;
   1:  PR[91,2] = PR[90,2] + -2.873;
   1:  PR[91,3] = PR[90,3] + 47.103;
   1:L PR[91] R[100]mm/sec CNT100;
   1:  PR[91,1] = PR[90,1] + -85.931;
   1:  PR[91,2] = PR[90,2] + -3.624;
   1:  PR[91,3] = PR[90,3] + 47.110;
   1:L PR[91] R[100]mm/sec CNT100;
   1:  PR[91,1] = PR[90,1] + -85.808;
   1:  PR[91,2] = PR[90,2] + -4.748;
   1:  PR[91,3] = PR[90,3] + 47.112;
   1:L PR[91] R[100]mm/sec CNT100;
   1:  PR[91,1] = PR[90,1] + -84.869;
   1:  PR[91,2] = PR[90,2] + -7.478;
   1:  PR[91,3] = PR[90,3] + 47.115;
   1:L PR[91] R[100]mm/sec CNT100;
   1:  PR[91,1] = PR[90,1] + -84.481;
   1:  PR[91,2] = PR[90,2] + -8.624;
   1:  PR[91,3] = PR[90,3] + 47.124;
   1:L PR[91] R[100]mm/sec CNT100;
   1:  PR[91,1] = PR[90,1] + -82.314;
   1:  PR[91,2] = PR[90,2] + -12.201;
   1:  PR[91,3] = PR[90,3] + 47.128;
   1:L PR[91] R[100]mm/sec CNT100;
   1:  PR[91,1] = PR[90,1] + -80.724;
   1:  PR[91,2] = PR[90,2] + -13.888;
   1:  PR[91,3] = PR[90,3] + 47.140;
   1:L PR[91] R[100]mm/sec CNT100;
   1:  PR[91,1] = PR[90,1] + -79.369;
   1:  PR[91,2] = PR[90,2] + -15.355;
   1:  PR[91,3] = PR[90,3] + 47.147;
   1:L PR[91] R[100]mm/sec CNT100;
   1:  PR[91,1] = PR[90,1] + -77.866;
   1:  PR[91,2] = PR[90,2] + -16.413;
   1:  PR[91,3] = PR[90,3] + 47.153;
   1:L PR[91] R[100]mm/sec CNT100;
   1:  PR[91,1] = PR[90,1] + -75.749;
   1:  PR[91,2] = PR[90,2] + -17.942;
   1:  PR[91,3] = PR[90,3] + 47.159;
   1:L PR[91] R[100]mm/sec CNT100;
   1:  PR[91,1] = PR[90,1] + -74.639;
   1:  PR[91,2] = PR[90,2] + -18.436;
   1:  PR[91,3] = PR[90,3] + 47.167;
   1:L PR[91] R[100]mm/sec CNT100;
   1:  PR[91,1] = PR[90,1] + -71.569;
   1:  PR[91,2] = PR[90,2] + -19.854;
   1:  PR[91,3] = PR[90,3] + 47.171;
   1:L PR[91] R[100]mm/sec CNT100;
   1:  PR[91,1] = PR[90,1] + -67.016;
   1:  PR[91,2] = PR[90,2] + -20.972;
   1:  PR[91,3] = PR[90,3] + 47.181;
   1:L PR[91] R[100]mm/sec CNT100;
   1:  PR[91,1] = PR[90,1] + -66.739;
   1:  PR[91,2] = PR[90,2] + -21.022;
   1:  PR[91,3] = PR[90,3] + 47.195;
   1:L PR[91] R[100]mm/sec CNT100;
   1:  PR[91,1] = PR[90,1] + -62.627;
   1:  PR[91,2] = PR[90,2] + -21.296;
   1:  PR[91,3] = PR[90,3] + 47.196;
   1:L PR[91] R[100]mm/sec CNT100;
   1:  PR[91,1] = PR[90,1] + -60.642;
   1:  PR[91,2] = PR[90,2] + -21.279;
   1:  PR[91,3] = PR[90,3] + 47.208;
   1:L PR[91] R[100]mm/sec CNT100;
   1:  PR[91,1] = PR[90,1] + -58.114;
   1:  PR[91,2] = PR[90,2] + -21.005;
   1:  PR[91,3] = PR[90,3] + 47.214;
   1:L PR[91] R[100]mm/sec CNT100;
   1:  PR[91,1] = PR[90,1] + -54.135;
   1:  PR[91,2] = PR[90,2] + -20.217;
   1:  PR[91,3] = PR[90,3] + 47.222;
   1:L PR[91] R[100]mm/sec CNT100;
   1:  PR[91,1] = PR[90,1] + -53.566;
   1:  PR[91,2] = PR[90,2] + -20.048;
   1:  PR[91,3] = PR[90,3] + 47.234;
   1:L PR[91] R[100]mm/sec CNT100;
   1:  PR[91,1] = PR[90,1] + -51.802;
   1:  PR[91,2] = PR[90,2] + -19.318;
   1:  PR[91,3] = PR[90,3] + 47.236;
   1:L PR[91] R[100]mm/sec CNT100;
   1:  PR[91,1] = PR[90,1] + -48.191;
   1:  PR[91,2] = PR[90,2] + -18.044;
   1:  PR[91,3] = PR[90,3] + 47.242;
   1:L PR[91] R[100]mm/sec CNT100;
   1:  PR[91,1] = PR[90,1] + -45.646;
   1:  PR[91,2] = PR[90,2] + -16.563;
   1:  PR[91,3] = PR[90,3] + 47.254;
   1:L PR[91] R[100]mm/sec CNT100;
   1:  PR[91,1] = PR[90,1] + -43.170;
   1:  PR[91,2] = PR[90,2] + -15.082;
   1:  PR[91,3] = PR[90,3] + 47.263;
   1:L PR[91] R[100]mm/sec CNT100;
   1:  PR[91,1] = PR[90,1] + -39.968;
   1:  PR[91,2] = PR[90,2] + -12.061;
   1:  PR[91,3] = PR[90,3] + 47.271;
   1:L PR[91] R[100]mm/sec CNT100;
   1:  PR[91,1] = PR[90,1] + -37.341;
   1:  PR[91,2] = PR[90,2] + -9.969;
   1:  PR[91,3] = PR[90,3] + 47.285;
   1:L PR[91] R[100]mm/sec CNT100;
   1:  PR[91,1] = PR[90,1] + -35.526;
   1:  PR[91,2] = PR[90,2] + -12.497;
   1:  PR[91,3] = PR[90,3] + 47.295;
   1:L PR[91] R[100]mm/sec CNT100;
   1:  PR[91,1] = PR[90,1] + -32.447;
   1:  PR[91,2] = PR[90,2] + -15.896;
   1:  PR[91,3] = PR[90,3] + 47.304;
   1:L PR[91] R[100]mm/sec CNT100;
   1:  PR[91,1] = PR[90,1] + -28.706;
   1:  PR[91,2] = PR[90,2] + -18.547;
   1:  PR[91,3] = PR[90,3] + 47.318;
   1:L PR[91] R[100]mm/sec CNT100;
   1:  PR[91,1] = PR[90,1] + -28.569;
   1:  PR[91,2] = PR[90,2] + -18.621;
   1:  PR[91,3] = PR[90,3] + 47.332;
   1:L PR[91] R[100]mm/sec CNT100;
   1:  PR[91,1] = PR[90,1] + -24.504;
   1:  PR[91,2] = PR[90,2] + -20.366;
   1:L PR[91] R[100]mm/sec CNT100;
   1:  PR[91,1] = PR[90,1] + -23.707;
   1:  PR[91,2] = PR[90,2] + -20.596;
   1:  PR[91,3] = PR[90,3] + 47.346;
   1:L PR[91] R[100]mm/sec CNT100;
   1:  PR[91,1] = PR[90,1] + -19.952;
   1:  PR[91,2] = PR[90,2] + -21.350;
   1:  PR[91,3] = PR[90,3] + 47.348;
   1:L PR[91] R[100]mm/sec CNT100;
   1:  PR[91,1] = PR[90,1] + -18.314;
   1:  PR[91,2] = PR[90,2] + -21.465;
   1:  PR[91,3] = PR[90,3] + 47.360;
   1:L PR[91] R[100]mm/sec CNT100;
   1:  PR[91,1] = PR[90,1] + -15.225;
   1:  PR[91,2] = PR[90,2] + -21.436;
   1:  PR[91,3] = PR[90,3] + 47.365;
   1:L PR[91] R[100]mm/sec CNT100;
   1:  PR[91,1] = PR[90,1] + -12.689;
   1:  PR[91,2] = PR[90,2] + -21.073;
   1:  PR[91,3] = PR[90,3] + 47.374;
   1:L PR[91] R[100]mm/sec CNT100;
   1:  PR[91,1] = PR[90,1] + -10.510;
   1:  PR[91,2] = PR[90,2] + -20.589;
   1:  PR[91,3] = PR[90,3] + 47.382;
   1:L PR[91] R[100]mm/sec CNT100;
   1:  PR[91,1] = PR[90,1] + -7.211;
   1:  PR[91,2] = PR[90,2] + -19.348;
   1:  PR[91,3] = PR[90,3] + 47.389;
   1:L PR[91] R[100]mm/sec CNT100;
   1:  PR[91,1] = PR[90,1] + -6.016;
   1:  PR[91,2] = PR[90,2] + -18.795;
   1:  PR[91,3] = PR[90,3] + 47.400;
   1:L PR[91] R[100]mm/sec CNT100;
   1:  PR[91,1] = PR[90,1] + -2.299;
   1:  PR[91,2] = PR[90,2] + -16.339;
   1:  PR[91,3] = PR[90,3] + 47.404;
   1:L PR[91] R[100]mm/sec CNT100;
   1:  PR[91,1] = PR[90,1] + -1.963;
   1:  PR[91,2] = PR[90,2] + -16.081;
   1:  PR[91,3] = PR[90,3] + 47.417;
   1:L PR[91] R[100]mm/sec CNT100;
   1:  PR[91,1] = PR[90,1] + 0.977;
   1:  PR[91,2] = PR[90,2] + -12.930;
   1:  PR[91,3] = PR[90,3] + 47.418;
   1:L PR[91] R[100]mm/sec CNT100;
   1:  PR[91,1] = PR[90,1] + 3.282;
   1:  PR[91,2] = PR[90,2] + -10.628;
   1:  PR[91,3] = PR[90,3] + 47.431;
   1:L PR[91] R[100]mm/sec CNT100;
   1:  PR[91,1] = PR[90,1] + 5.560;
   1:  PR[91,2] = PR[90,2] + -13.885;
   1:  PR[91,3] = PR[90,3] + 47.441;
   1:L PR[91] R[100]mm/sec CNT100;
   1:  PR[91,1] = PR[90,1] + 8.911;
   1:  PR[91,2] = PR[90,2] + -17.416;
   1:  PR[91,3] = PR[90,3] + 47.453;
   1:L PR[91] R[100]mm/sec CNT100;
   1:  PR[91,1] = PR[90,1] + 9.527;
   1:  PR[91,2] = PR[90,2] + -17.884;
   1:  PR[91,3] = PR[90,3] + 47.468;
   1:L PR[91] R[100]mm/sec CNT100;
   1:  PR[91,1] = PR[90,1] + 13.497;
   1:  PR[91,2] = PR[90,2] + -20.358;
   1:  PR[91,3] = PR[90,3] + 47.470;
   1:L PR[91] R[100]mm/sec CNT100;
   1:  PR[91,1] = PR[90,1] + 14.380;
   1:  PR[91,2] = PR[90,2] + -20.719;
   1:  PR[91,3] = PR[90,3] + 47.485;
   1:L PR[91] R[100]mm/sec CNT100;
   1:  PR[91,1] = PR[90,1] + 18.663;
   1:  PR[91,2] = PR[90,2] + -22.075;
   1:  PR[91,3] = PR[90,3] + 47.487;
   1:L PR[91] R[100]mm/sec CNT100;
   1:  PR[91,1] = PR[90,1] + 19.804;
   1:  PR[91,2] = PR[90,2] + -22.221;
   1:  PR[91,3] = PR[90,3] + 47.501;
   1:L PR[91] R[100]mm/sec CNT100;
   1:  PR[91,1] = PR[90,1] + 24.089;
   1:  PR[91,2] = PR[90,2] + -22.467;
   1:  PR[91,3] = PR[90,3] + 47.505;
   1:L PR[91] R[100]mm/sec CNT100;
   1:  PR[91,1] = PR[90,1] + 25.426;
   1:  PR[91,2] = PR[90,2] + -22.289;
   1:  PR[91,3] = PR[90,3] + 47.518;
   1:L PR[91] R[100]mm/sec CNT100;
   1:  PR[91,1] = PR[90,1] + 29.443;
   1:  PR[91,2] = PR[90,2] + -21.511;
   1:  PR[91,3] = PR[90,3] + 47.522;
   1:L PR[91] R[100]mm/sec CNT100;
   1:  PR[91,1] = PR[90,1] + 30.864;
   1:  PR[91,2] = PR[90,2] + -20.925;
   1:  PR[91,3] = PR[90,3] + 47.534;
   1:L PR[91] R[100]mm/sec CNT100;
   1:  PR[91,1] = PR[90,1] + 34.392;
   1:  PR[91,2] = PR[90,2] + -19.268;
   1:  PR[91,3] = PR[90,3] + 47.539;
   1:L PR[91] R[100]mm/sec CNT100;
   1:  PR[91,1] = PR[90,1] + 35.893;
   1:  PR[91,2] = PR[90,2] + -18.129;
   1:  PR[91,3] = PR[90,3] + 47.551;
   1:L PR[91] R[100]mm/sec CNT100;
   1:  PR[91,1] = PR[90,1] + 36.272;
   1:  PR[91,2] = PR[90,2] + -17.920;
   1:  PR[91,3] = PR[90,3] + 47.556;
   1:L PR[91] R[100]mm/sec CNT100;
   1:  PR[91,1] = PR[90,1] + 36.696;
   1:  PR[91,2] = PR[90,2] + -17.632;
   1:  PR[91,3] = PR[90,3] + 47.558;
   1:L PR[91] R[100]mm/sec CNT100;
   1:  PR[91,1] = PR[90,1] + 38.129;
   1:  PR[91,2] = PR[90,2] + -16.301;
   1:  PR[91,3] = PR[90,3] + 47.559;
   1:L PR[91] R[100]mm/sec CNT100;
   1:  PR[91,1] = PR[90,1] + 40.873;
   1:  PR[91,2] = PR[90,2] + -18.006;
   1:  PR[91,3] = PR[90,3] + 47.565;
   1:L PR[91] R[100]mm/sec CNT100;
   1:  PR[91,1] = PR[90,1] + 43.257;
   1:  PR[91,2] = PR[90,2] + -19.203;
   1:  PR[91,3] = PR[90,3] + 47.575;
   1:L PR[91] R[100]mm/sec CNT100;
   1:  PR[91,1] = PR[90,1] + 47.114;
   1:  PR[91,2] = PR[90,2] + -20.615;
   1:  PR[91,3] = PR[90,3] + 47.583;
   1:L PR[91] R[100]mm/sec CNT100;
   1:  PR[91,1] = PR[90,1] + 48.535;
   1:  PR[91,2] = PR[90,2] + -21.211;
   1:  PR[91,3] = PR[90,3] + 47.595;
   1:L PR[91] R[100]mm/sec CNT100;
   1:  PR[91,1] = PR[90,1] + 49.240;
   1:  PR[91,2] = PR[90,2] + -21.483;
   1:  PR[91,3] = PR[90,3] + 47.600;
   1:L PR[91] R[100]mm/sec CNT100;
   1:  PR[91,1] = PR[90,1] + 52.855;
   1:  PR[91,2] = PR[90,2] + -22.219;
   1:  PR[91,3] = PR[90,3] + 47.602;
   1:L PR[91] R[100]mm/sec CNT100;
   1:  PR[91,1] = PR[90,1] + 56.499;
   1:  PR[91,2] = PR[90,2] + -22.877;
   1:  PR[91,3] = PR[90,3] + 47.613;
   1:L PR[91] R[100]mm/sec CNT100;
   1:  PR[91,1] = PR[90,1] + 57.329;
   1:  PR[91,2] = PR[90,2] + -22.892;
   1:  PR[91,3] = PR[90,3] + 47.625;
   1:L PR[91] R[100]mm/sec CNT100;
   1:  PR[91,1] = PR[90,1] + 59.245;
   1:  PR[91,2] = PR[90,2] + -22.894;
   1:  PR[91,3] = PR[90,3] + 47.627;
   1:L PR[91] R[100]mm/sec CNT100;
   1:  PR[91,1] = PR[90,1] + 62.437;
   1:  PR[91,2] = PR[90,2] + -22.950;
   1:  PR[91,3] = PR[90,3] + 47.633;
   1:L PR[91] R[100]mm/sec CNT100;
   1:  PR[91,1] = PR[90,1] + 63.971;
   1:  PR[91,2] = PR[90,2] + -22.810;
   1:  PR[91,3] = PR[90,3] + 47.643;
   1:L PR[91] R[100]mm/sec CNT100;
   1:  PR[91,1] = PR[90,1] + 67.531;
   1:  PR[91,2] = PR[90,2] + -22.193;
   1:  PR[91,3] = PR[90,3] + 47.647;
   1:L PR[91] R[100]mm/sec CNT100;
   1:  PR[91,1] = PR[90,1] + 71.379;
   1:  PR[91,2] = PR[90,2] + -21.037;
   1:  PR[91,3] = PR[90,3] + 47.658;
   1:L PR[91] R[100]mm/sec CNT100;
   1:  PR[91,1] = PR[90,1] + 72.585;
   1:  PR[91,2] = PR[90,2] + -20.581;
   1:  PR[91,3] = PR[90,3] + 47.670;
   1:L PR[91] R[100]mm/sec CNT100;
   1:  PR[91,1] = PR[90,1] + 76.546;
   1:  PR[91,2] = PR[90,2] + -18.427;
   1:  PR[91,3] = PR[90,3] + 47.674;
   1:L PR[91] R[100]mm/sec CNT100;
   1:  PR[91,1] = PR[90,1] + 77.350;
   1:  PR[91,2] = PR[90,2] + -17.983;
   1:  PR[91,3] = PR[90,3] + 47.688;
   1:L PR[91] R[100]mm/sec CNT100;
   1:  PR[91,1] = PR[90,1] + 80.830;
   1:  PR[91,2] = PR[90,2] + -14.874;
   1:  PR[91,3] = PR[90,3] + 47.691;
   1:L PR[91] R[100]mm/sec CNT100;
   1:  PR[91,1] = PR[90,1] + 81.434;
   1:  PR[91,2] = PR[90,2] + -14.276;
   1:  PR[91,3] = PR[90,3] + 47.705;
   1:L PR[91] R[100]mm/sec CNT100;
   1:  PR[91,1] = PR[90,1] + 83.564;
   1:  PR[91,2] = PR[90,2] + -11.223;
   1:  PR[91,3] = PR[90,3] + 47.708;
   1:L PR[91] R[100]mm/sec CNT100;
   1:  PR[91,1] = PR[90,1] + 84.331;
   1:  PR[91,2] = PR[90,2] + -10.033;
   1:  PR[91,3] = PR[90,3] + 47.719;
   1:L PR[91] R[100]mm/sec CNT100;
   1:  PR[91,1] = PR[90,1] + 85.460;
   1:  PR[91,2] = PR[90,2] + -7.113;
   1:  PR[91,3] = PR[90,3] + 47.723;
   1:L PR[91] R[100]mm/sec CNT100;
   1:  PR[91,1] = PR[90,1] + 86.056;
   1:  PR[91,2] = PR[90,2] + -5.467;
   1:  PR[91,3] = PR[90,3] + 47.733;
   1:L PR[91] R[100]mm/sec CNT100;
   1:  PR[91,1] = PR[90,1] + 86.291;
   1:  PR[91,2] = PR[90,2] + -3.478;
   1:  PR[91,3] = PR[90,3] + 47.738;
   1:L PR[91] R[100]mm/sec CNT100;
   1:  PR[91,1] = PR[90,1] + 86.360;
   1:  PR[91,2] = PR[90,2] + -3.161;
   1:  PR[91,3] = PR[90,3] + 47.744;
   1:L PR[91] R[100]mm/sec CNT100;
   1:  PR[91,1] = PR[90,1] + 86.660;
   1:  PR[91,2] = PR[90,2] + -0.738;
   1:  PR[91,3] = PR[90,3] + 47.745;
   1:L PR[91] R[100]mm/sec CNT100;
   1:  PR[91,1] = PR[90,1] + 86.405;
   1:  PR[91,2] = PR[90,2] + 1.185;
   1:  PR[91,3] = PR[90,3] + 47.752;
   1:L PR[91] R[100]mm/sec CNT100;
   1:  PR[91,1] = PR[90,1] + 86.057;
   1:  PR[91,2] = PR[90,2] + 4.003;
   1:  PR[91,3] = PR[90,3] + 47.758;
   1:L PR[91] R[100]mm/sec CNT100;
   1:  PR[91,1] = PR[90,1] + 85.460;
   1:  PR[91,2] = PR[90,2] + 5.654;
   1:  PR[91,3] = PR[90,3] + 47.767;
   1:L PR[91] R[100]mm/sec CNT100;
   1:  PR[91,1] = PR[90,1] + 84.331;
   1:  PR[91,2] = PR[90,2] + 8.574;
   1:  PR[91,3] = PR[90,3] + 47.772;
   1:L PR[91] R[100]mm/sec CNT100;
   1:  PR[91,1] = PR[90,1] + 83.564;
   1:  PR[91,2] = PR[90,2] + 9.764;
   1:  PR[91,3] = PR[90,3] + 47.782;
   1:L PR[91] R[100]mm/sec CNT100;
   1:  PR[91,1] = PR[90,1] + 81.434;
   1:  PR[91,2] = PR[90,2] + 12.817;
   1:  PR[91,3] = PR[90,3] + 47.786;
   1:L PR[91] R[100]mm/sec CNT100;
   1:  PR[91,1] = PR[90,1] + 80.831;
   1:  PR[91,2] = PR[90,2] + 13.415;
   1:  PR[91,3] = PR[90,3] + 47.797;
   1:L PR[91] R[100]mm/sec CNT100;
   1:  PR[91,1] = PR[90,1] + 77.350;
   1:  PR[91,2] = PR[90,2] + 16.524;
   1:  PR[91,3] = PR[90,3] + 47.800;
   1:L PR[91] R[100]mm/sec CNT100;
   1:  PR[91,1] = PR[90,1] + 76.545;
   1:  PR[91,2] = PR[90,2] + 16.968;
   1:  PR[91,3] = PR[90,3] + 47.814;
   1:L PR[91] R[100]mm/sec CNT100;
   1:  PR[91,1] = PR[90,1] + 72.579;
   1:  PR[91,2] = PR[90,2] + 19.125;
   1:  PR[91,3] = PR[90,3] + 47.817;
   1:L PR[91] R[100]mm/sec CNT100;
   1:  PR[91,1] = PR[90,1] + 71.361;
   1:  PR[91,2] = PR[90,2] + 19.584;
   1:  PR[91,3] = PR[90,3] + 47.830;
   1:L PR[91] R[100]mm/sec CNT100;
   1:  PR[91,1] = PR[90,1] + 67.510;
   1:  PR[91,2] = PR[90,2] + 20.740;
   1:  PR[91,3] = PR[90,3] + 47.834;
   1:L PR[91] R[100]mm/sec CNT100;
   1:  PR[91,1] = PR[90,1] + 63.908;
   1:  PR[91,2] = PR[90,2] + 21.358;
   1:  PR[91,3] = PR[90,3] + 47.846;
   1:L PR[91] R[100]mm/sec CNT100;
   1:  PR[91,1] = PR[90,1] + 62.391;
   1:  PR[91,2] = PR[90,2] + 21.496;
   1:  PR[91,3] = PR[90,3] + 47.858;
   1:L PR[91] R[100]mm/sec CNT100;
   1:  PR[91,1] = PR[90,1] + 59.254;
   1:  PR[91,2] = PR[90,2] + 21.433;
   1:  PR[91,3] = PR[90,3] + 47.862;
   1:L PR[91] R[100]mm/sec CNT100;
   1:  PR[91,1] = PR[90,1] + 56.424;
   1:  PR[91,2] = PR[90,2] + 21.410;
   1:  PR[91,3] = PR[90,3] + 47.872;
   1:L PR[91] R[100]mm/sec CNT100;
   1:  PR[91,1] = PR[90,1] + 52.832;
   1:  PR[91,2] = PR[90,2] + 20.749;
   1:  PR[91,3] = PR[90,3] + 47.880;
   1:L PR[91] R[100]mm/sec CNT100;
   1:  PR[91,1] = PR[90,1] + 49.256;
   1:  PR[91,2] = PR[90,2] + 20.029;
   1:  PR[91,3] = PR[90,3] + 47.891;
   1:L PR[91] R[100]mm/sec CNT100;
   1:  PR[91,1] = PR[90,1] + 48.551;
   1:  PR[91,2] = PR[90,2] + 19.754;
   1:  PR[91,3] = PR[90,3] + 47.902;
   1:L PR[91] R[100]mm/sec CNT100;
   1:  PR[91,1] = PR[90,1] + 47.111;
   1:  PR[91,2] = PR[90,2] + 19.153;
   1:  PR[91,3] = PR[90,3] + 47.905;
   1:L PR[91] R[100]mm/sec CNT100;
   1:  PR[91,1] = PR[90,1] + 43.277;
   1:  PR[91,2] = PR[90,2] + 17.755;
   1:  PR[91,3] = PR[90,3] + 47.909;
   1:L PR[91] R[100]mm/sec CNT100;
   1:  PR[91,1] = PR[90,1] + 40.899;
   1:  PR[91,2] = PR[90,2] + 16.560;
   1:  PR[91,3] = PR[90,3] + 47.922;
   1:L PR[91] R[100]mm/sec CNT100;
   1:  PR[91,1] = PR[90,1] + 38.085;
   1:  PR[91,2] = PR[90,2] + 14.788;
   1:  PR[91,3] = PR[90,3] + 47.930;
   1:L PR[91] R[100]mm/sec CNT100;
   1:  PR[91,1] = PR[90,1] + 36.629;
   1:  PR[91,2] = PR[90,2] + 16.231;
   1:  PR[91,3] = PR[90,3] + 47.940;
   1:L PR[91] R[100]mm/sec CNT100;
   1:  PR[91,1] = PR[90,1] + 36.265;
   1:  PR[91,2] = PR[90,2] + 16.506;
   1:  PR[91,3] = PR[90,3] + 47.946;
   1:L PR[91] R[100]mm/sec CNT100;
   1:  PR[91,1] = PR[90,1] + 34.990;
   1:  PR[91,2] = PR[90,2] + 17.425;
   1:  PR[91,3] = PR[90,3] + 47.947;
   1:L PR[91] R[100]mm/sec CNT100;
   1:  PR[91,1] = PR[90,1] + 34.440;
   1:  PR[91,2] = PR[90,2] + 17.788;
   1:  PR[91,3] = PR[90,3] + 47.952;
   1:L PR[91] R[100]mm/sec CNT100;
   1:  PR[91,1] = PR[90,1] + 30.855;
   1:  PR[91,2] = PR[90,2] + 19.472;
   1:  PR[91,3] = PR[90,3] + 47.954;
   1:L PR[91] R[100]mm/sec CNT100;
   1:  PR[91,1] = PR[90,1] + 29.435;
   1:  PR[91,2] = PR[90,2] + 20.055;
   1:  PR[91,3] = PR[90,3] + 47.966;
   1:L PR[91] R[100]mm/sec CNT100;
   1:  PR[91,1] = PR[90,1] + 25.421;
   1:  PR[91,2] = PR[90,2] + 20.833;
   1:  PR[91,3] = PR[90,3] + 47.971;
   1:L PR[91] R[100]mm/sec CNT100;
   1:  PR[91,1] = PR[90,1] + 24.085;
   1:  PR[91,2] = PR[90,2] + 21.008;
   1:  PR[91,3] = PR[90,3] + 47.983;
   1:L PR[91] R[100]mm/sec CNT100;
   1:  PR[91,1] = PR[90,1] + 19.803;
   1:  PR[91,2] = PR[90,2] + 20.763;
   1:  PR[91,3] = PR[90,3] + 47.987;
   1:L PR[91] R[100]mm/sec CNT100;
   1:  PR[91,1] = PR[90,1] + 18.663;
   1:  PR[91,2] = PR[90,2] + 20.616;
   1:  PR[91,3] = PR[90,3] + 48.000;
   1:L PR[91] R[100]mm/sec CNT100;
   1:  PR[91,1] = PR[90,1] + 14.383;
   1:  PR[91,2] = PR[90,2] + 19.262;
   1:  PR[91,3] = PR[90,3] + 48.004;
   1:L PR[91] R[100]mm/sec CNT100;
   1:  PR[91,1] = PR[90,1] + 13.501;
   1:  PR[91,2] = PR[90,2] + 18.901;
   1:  PR[91,3] = PR[90,3] + 48.017;
   1:L PR[91] R[100]mm/sec CNT100;
   1:  PR[91,1] = PR[90,1] + 9.533;
   1:  PR[91,2] = PR[90,2] + 16.430;
   1:  PR[91,3] = PR[90,3] + 48.020;
   1:L PR[91] R[100]mm/sec CNT100;
   1:  PR[91,1] = PR[90,1] + 8.917;
   1:  PR[91,2] = PR[90,2] + 15.962;
   1:  PR[91,3] = PR[90,3] + 48.034;
   1:L PR[91] R[100]mm/sec CNT100;
   1:  PR[91,1] = PR[90,1] + 5.534;
   1:  PR[91,2] = PR[90,2] + 12.403;
   1:  PR[91,3] = PR[90,3] + 48.037;
   1:L PR[91] R[100]mm/sec CNT100;
   1:  PR[91,1] = PR[90,1] + 5.147;
   1:  PR[91,2] = PR[90,2] + 11.903;
   1:  PR[91,3] = PR[90,3] + 48.052;
   1:L PR[91] R[100]mm/sec CNT100;
   1:  PR[91,1] = PR[90,1] + 3.351;
   1:  PR[91,2] = PR[90,2] + 9.129;
   1:  PR[91,3] = PR[90,3] + 48.054;
   1:L PR[91] R[100]mm/sec CNT100;
   1:  PR[91,1] = PR[90,1] + 0.875;
   1:  PR[91,2] = PR[90,2] + 11.572;
   1:  PR[91,3] = PR[90,3] + 48.064;
   1:L PR[91] R[100]mm/sec CNT100;
   1:  PR[91,1] = PR[90,1] + -1.943;
   1:  PR[91,2] = PR[90,2] + 14.606;
   1:  PR[91,3] = PR[90,3] + 48.074;
   1:L PR[91] R[100]mm/sec CNT100;
   1:  PR[91,1] = PR[90,1] + -2.275;
   1:  PR[91,2] = PR[90,2] + 14.861;
   1:  PR[91,3] = PR[90,3] + 48.087;
   1:L PR[91] R[100]mm/sec CNT100;
   1:  PR[91,1] = PR[90,1] + -5.993;
   1:  PR[91,2] = PR[90,2] + 17.324;
   1:  PR[91,3] = PR[90,3] + 48.088;
   1:L PR[91] R[100]mm/sec CNT100;
   1:  PR[91,1] = PR[90,1] + -7.184;
   1:  PR[91,2] = PR[90,2] + 17.876;
   1:  PR[91,3] = PR[90,3] + 48.101;
   1:L PR[91] R[100]mm/sec CNT100;
   1:  PR[91,1] = PR[90,1] + -10.486;
   1:  PR[91,2] = PR[90,2] + 19.124;
   1:  PR[91,3] = PR[90,3] + 48.105;
   1:L PR[91] R[100]mm/sec CNT100;
   1:  PR[91,1] = PR[90,1] + -12.662;
   1:  PR[91,2] = PR[90,2] + 19.608;
   1:  PR[91,3] = PR[90,3] + 48.116;
   1:L PR[91] R[100]mm/sec CNT100;
   1:  PR[91,1] = PR[90,1] + -15.202;
   1:  PR[91,2] = PR[90,2] + 19.976;
   1:  PR[91,3] = PR[90,3] + 48.123;
   1:L PR[91] R[100]mm/sec CNT100;
   1:  PR[91,1] = PR[90,1] + -18.289;
   1:  PR[91,2] = PR[90,2] + 20.007;
   1:  PR[91,3] = PR[90,3] + 48.131;
   1:L PR[91] R[100]mm/sec CNT100;
   1:  PR[91,1] = PR[90,1] + -19.932;
   1:  PR[91,2] = PR[90,2] + 19.894;
   1:  PR[91,3] = PR[90,3] + 48.140;
   1:L PR[91] R[100]mm/sec CNT100;
   1:  PR[91,1] = PR[90,1] + -23.687;
   1:  PR[91,2] = PR[90,2] + 19.142;
   1:  PR[91,3] = PR[90,3] + 48.145;
   1:L PR[91] R[100]mm/sec CNT100;
   1:  PR[91,1] = PR[90,1] + -24.488;
   1:  PR[91,2] = PR[90,2] + 18.912;
   1:  PR[91,3] = PR[90,3] + 48.157;
   1:L PR[91] R[100]mm/sec CNT100;
   1:  PR[91,1] = PR[90,1] + -28.556;
   1:  PR[91,2] = PR[90,2] + 17.169;
   1:  PR[91,3] = PR[90,3] + 48.159;
   1:L PR[91] R[100]mm/sec CNT100;
   1:  PR[91,1] = PR[90,1] + -28.692;
   1:  PR[91,2] = PR[90,2] + 17.097;
   1:  PR[91,3] = PR[90,3] + 48.173;
   1:L PR[91] R[100]mm/sec CNT100;
   1:  PR[91,1] = PR[90,1] + -32.438;
   1:  PR[91,2] = PR[90,2] + 14.445;
   1:L PR[91] R[100]mm/sec CNT100;
   1:  PR[91,1] = PR[90,1] + -35.474;
   1:  PR[91,2] = PR[90,2] + 11.098;
   1:  PR[91,3] = PR[90,3] + 48.187;
   1:L PR[91] R[100]mm/sec CNT100;
   1:  PR[91,1] = PR[90,1] + -35.693;
   1:  PR[91,2] = PR[90,2] + 10.750;
   1:  PR[91,3] = PR[90,3] + 48.201;
   1:L PR[91] R[100]mm/sec CNT100;
   1:  PR[91,1] = PR[90,1] + -37.721;
   1:  PR[91,2] = PR[90,2] + 8.290;
   1:  PR[91,3] = PR[90,3] + 48.202;
   1:L PR[91] R[100]mm/sec CNT100;
   1:  PR[91,1] = PR[90,1] + -39.998;
   1:  PR[91,2] = PR[90,2] + 10.948;
   1:  PR[91,3] = PR[90,3] + 48.212;
   1:L PR[91] R[100]mm/sec CNT100;
   1:  PR[91,1] = PR[90,1] + -42.154;
   1:  PR[91,2] = PR[90,2] + 12.689;
   1:  PR[91,3] = PR[90,3] + 48.222;
   1:L PR[91] R[100]mm/sec CNT100;
   1:  PR[91,1] = PR[90,1] + -44.987;
   1:  PR[91,2] = PR[90,2] + 14.792;
   1:  PR[91,3] = PR[90,3] + 48.231;
   1:L PR[91] R[100]mm/sec CNT100;
   1:  PR[91,1] = PR[90,1] + -45.412;
   1:  PR[91,2] = PR[90,2] + 15.004;
   1:  PR[91,3] = PR[90,3] + 48.241;
   1:L PR[91] R[100]mm/sec CNT100;
   1:  PR[91,1] = PR[90,1] + -46.504;
   1:  PR[91,2] = PR[90,2] + 15.510;
   1:  PR[91,3] = PR[90,3] + 48.243;
   1:L PR[91] R[100]mm/sec CNT100;
   1:  PR[91,1] = PR[90,1] + -49.373;
   1:  PR[91,2] = PR[90,2] + 17.032;
   1:  PR[91,3] = PR[90,3] + 48.246;
   1:L PR[91] R[100]mm/sec CNT100;
   1:  PR[91,1] = PR[90,1] + -50.524;
   1:  PR[91,2] = PR[90,2] + 17.595;
   1:  PR[91,3] = PR[90,3] + 48.256;
   1:L PR[91] R[100]mm/sec CNT100;
   1:  PR[91,1] = PR[90,1] + -53.133;
   1:  PR[91,2] = PR[90,2] + 18.389;
   1:  PR[91,3] = PR[90,3] + 48.260;
   1:L PR[91] R[100]mm/sec CNT100;
   1:  PR[91,1] = PR[90,1] + -56.295;
   1:  PR[91,2] = PR[90,2] + 19.264;
   1:  PR[91,3] = PR[90,3] + 48.268;
   1:L PR[91] R[100]mm/sec CNT100;
   1:  PR[91,1] = PR[90,1] + -57.061;
   1:  PR[91,2] = PR[90,2] + 19.353;
   1:  PR[91,3] = PR[90,3] + 48.278;
   1:L PR[91] R[100]mm/sec CNT100;
   1:  PR[91,1] = PR[90,1] + -59.319;
   1:  PR[91,2] = PR[90,2] + 19.571;
   1:  PR[91,3] = PR[90,3] + 48.281;
   1:L PR[91] R[100]mm/sec CNT100;
   1:  PR[91,1] = PR[90,1] + -61.795;
   1:  PR[91,2] = PR[90,2] + 19.863;
   1:  PR[91,3] = PR[90,3] + 48.287;
   1:L PR[91] R[100]mm/sec CNT100;
   1:  PR[91] = PR[90];
   1:  PR[91,1] = PR[90,1] + -66.110;
   1:  PR[91,2] = PR[90,2] + 19.696;
   1:  PR[91,3] = PR[90,3] + 49.595;
   1:L PR[91] R[100]mm/sec CNT100;
   1:  PR[91,1] = PR[90,1] + -67.933;
   1:  PR[91,2] = PR[90,2] + 19.258;
   1:  PR[91,3] = PR[90,3] + 48.310;
   1:L PR[91] R[100]mm/sec CNT100;
   1:  PR[91,1] = PR[90,1] + -70.889;
   1:  PR[91,2] = PR[90,2] + 18.522;
   1:  PR[91,3] = PR[90,3] + 48.316;
   1:L PR[91] R[100]mm/sec CNT100;
   1:  PR[91,1] = PR[90,1] + -75.246;
   1:  PR[91,2] = PR[90,2] + 16.570;
   1:  PR[91,3] = PR[90,3] + 48.325;
   1:L PR[91] R[100]mm/sec CNT100;
   1:  PR[91,1] = PR[90,1] + -78.977;
   1:  PR[91,2] = PR[90,2] + 13.971;
   1:  PR[91,3] = PR[90,3] + 48.340;
   1:L PR[91] R[100]mm/sec CNT100;
   1:  PR[91,1] = PR[90,1] + -79.006;
   1:  PR[91,2] = PR[90,2] + 13.950;
   1:  PR[91,3] = PR[90,3] + 48.354;
   1:L PR[91] R[100]mm/sec CNT100;
   1:  PR[91,1] = PR[90,1] + -79.746;
   1:  PR[91,2] = PR[90,2] + 13.178;
   1:L PR[91] R[100]mm/sec CNT100;
   1:  PR[91,1] = PR[90,1] + -81.924;
   1:  PR[91,2] = PR[90,2] + 10.806;
   1:  PR[91,3] = PR[90,3] + 48.357;
   1:L PR[91] R[100]mm/sec CNT100;
   1:  PR[91,1] = PR[90,1] + -84.066;
   1:  PR[91,2] = PR[90,2] + 7.208;
   1:  PR[91,3] = PR[90,3] + 48.367;
   1:L PR[91] R[100]mm/sec CNT100;
   1:  PR[91,1] = PR[90,1] + -85.377;
   1:  PR[91,2] = PR[90,2] + 3.313;
   1:  PR[91,3] = PR[90,3] + 48.379;
   1:L PR[91] R[100]mm/sec CNT100;
   1:  PR[91,1] = PR[90,1] + -85.479;
   1:  PR[91,2] = PR[90,2] + 2.392;
   1:  PR[91,3] = PR[90,3] + 48.392;
   1:L PR[91] R[100]mm/sec CNT100;
   1:  PR[91,1] = PR[90,1] + -85.589;
   1:  PR[91,2] = PR[90,2] + 1.818;
   1:  PR[91,3] = PR[90,3] + 48.395;
   1:L PR[91] R[100]mm/sec CNT100;
   1:  PR[91,1] = PR[90,1] + -85.868;
   1:  PR[91,2] = PR[90,2] + -0.728;
   1:  PR[91,3] = PR[90,3] + 48.397;
   1:L PR[91] R[100]mm/sec CNT100;
   1:  PR[91,1] = PR[90,1] + -85.717;
   1:  PR[91,2] = PR[90,2] + -2.089;
   1:  PR[91,3] = PR[90,3] + 48.404;
   1:L PR[91] R[100]mm/sec CNT100;
   1:  PR[91,1] = PR[90,1] + -85.488;
   1:  PR[91,2] = PR[90,2] + -3.143;
   1:  PR[91,3] = PR[90,3] + 48.408;
   1:L PR[91] R[100]mm/sec CNT100;
   1:  PR[91,1] = PR[90,1] + -85.309;
   1:  PR[91,2] = PR[90,2] + -4.767;
   1:  PR[91,3] = PR[90,3] + 48.412;
   1:L PR[91] R[100]mm/sec CNT100;
   1:  PR[91,1] = PR[90,1] + -84.526;
   1:  PR[91,2] = PR[90,2] + -7.046;
   1:  PR[91,3] = PR[90,3] + 48.417;
   1:L PR[91] R[100]mm/sec CNT100;
   1:  PR[91,1] = PR[90,1] + -83.977;
   1:  PR[91,2] = PR[90,2] + -8.663;
   1:  PR[91,3] = PR[90,3] + 48.424;
   1:L PR[91] R[100]mm/sec CNT100;
   1:  PR[91,1] = PR[90,1] + -81.803;
   1:  PR[91,2] = PR[90,2] + -12.259;
   1:  PR[91,3] = PR[90,3] + 48.429;
   1:L PR[91] R[100]mm/sec CNT100;
   1:  PR[91,1] = PR[90,1] + -80.550;
   1:  PR[91,2] = PR[90,2] + -13.590;
   1:  PR[91,3] = PR[90,3] + 48.442;
   1:L PR[91] R[100]mm/sec CNT100;
   1:  PR[91,1] = PR[90,1] + -78.847;
   1:  PR[91,2] = PR[90,2] + -15.432;
   1:  PR[91,3] = PR[90,3] + 48.447;
   1:L PR[91] R[100]mm/sec CNT100;
   1:  PR[91,1] = PR[90,1] + -77.758;
   1:  PR[91,2] = PR[90,2] + -16.199;
   1:  PR[91,3] = PR[90,3] + 48.455;
   1:L PR[91] R[100]mm/sec CNT100;
   1:  PR[91,1] = PR[90,1] + -75.202;
   1:  PR[91,2] = PR[90,2] + -18.044;
   1:  PR[91,3] = PR[90,3] + 48.459;
   1:L PR[91] R[100]mm/sec CNT100;
   1:  PR[91,1] = PR[90,1] + -71.014;
   1:  PR[91,2] = PR[90,2] + -19.966;
   1:  PR[91,3] = PR[90,3] + 48.469;
   1:L PR[91] R[100]mm/sec CNT100;
   1:  PR[91,1] = PR[90,1] + -66.685;
   1:  PR[91,2] = PR[90,2] + -21.026;
   1:  PR[91,3] = PR[90,3] + 48.483;
   1:L PR[91] R[100]mm/sec CNT100;
   1:  PR[91,1] = PR[90,1] + -65.560;
   1:  PR[91,2] = PR[90,2] + -21.227;
   1:  PR[91,3] = PR[90,3] + 48.496;
   1:L PR[91] R[100]mm/sec CNT100;
   1:  PR[91,1] = PR[90,1] + -62.263;
   1:  PR[91,2] = PR[90,2] + -21.447;
   1:  PR[91,3] = PR[90,3] + 48.500;
   1:L PR[91] R[100]mm/sec CNT100;
   1:  PR[91,1] = PR[90,1] + -59.310;
   1:  PR[91,2] = PR[90,2] + -21.421;
   1:  PR[91,3] = PR[90,3] + 48.510;
   1:L PR[91] R[100]mm/sec CNT100;
   1:  PR[91,1] = PR[90,1] + -57.693;
   1:  PR[91,2] = PR[90,2] + -21.246;
   1:  PR[91,3] = PR[90,3] + 48.519;
   1:L PR[91] R[100]mm/sec CNT100;
   1:  PR[91,1] = PR[90,1] + -53.274;
   1:  PR[91,2] = PR[90,2] + -20.370;
   1:  PR[91,3] = PR[90,3] + 48.524;
   1:L PR[91] R[100]mm/sec CNT100;
   1:  PR[91,1] = PR[90,1] + -52.746;
   1:  PR[91,2] = PR[90,2] + -20.286;
   1:  PR[91,3] = PR[90,3] + 48.537;
   1:L PR[91] R[100]mm/sec CNT100;
   1:  PR[91,1] = PR[90,1] + -46.999;
   1:  PR[91,2] = PR[90,2] + -18.265;
   1:  PR[91,3] = PR[90,3] + 48.539;
   1:L PR[91] R[100]mm/sec CNT100;
   1:  PR[91,1] = PR[90,1] + -41.895;
   1:  PR[91,2] = PR[90,2] + -15.287;
   1:  PR[91,3] = PR[90,3] + 48.557;
   1:L PR[91] R[100]mm/sec CNT100;
   1:  PR[91,1] = PR[90,1] + -41.329;
   1:  PR[91,2] = PR[90,2] + -14.753;
   1:  PR[91,3] = PR[90,3] + 48.575;
   1:L PR[91] R[100]mm/sec CNT100;
   1:  PR[91,1] = PR[90,1] + -36.700;
   1:  PR[91,2] = PR[90,2] + -11.068;
   1:  PR[91,3] = PR[90,3] + 48.578;
   1:L PR[91] R[100]mm/sec CNT100;
   1:  PR[91,1] = PR[90,1] + -34.175;
   1:  PR[91,2] = PR[90,2] + -13.637;
   1:  PR[91,3] = PR[90,3] + 48.596;
   1:L PR[91] R[100]mm/sec CNT100;
   1:  PR[91,1] = PR[90,1] + -34.248;
   1:  PR[91,2] = PR[90,2] + -13.726;
   1:  PR[91,3] = PR[90,3] + 48.606;
   1:L PR[91] R[100]mm/sec CNT100;
   1:  PR[91,1] = PR[90,1] + -33.501;
   1:  PR[91,2] = PR[90,2] + -14.564;
   1:  PR[91,3] = PR[90,3] + 48.607;
   1:L PR[91] R[100]mm/sec CNT100;
   1:  PR[91,1] = PR[90,1] + -32.265;
   1:  PR[91,2] = PR[90,2] + -15.887;
   1:  PR[91,3] = PR[90,3] + 48.610;
   1:L PR[91] R[100]mm/sec CNT100;
   1:  PR[91,1] = PR[90,1] + -32.108;
   1:  PR[91,2] = PR[90,2] + -16.017;
   1:  PR[91,3] = PR[90,3] + 48.616;
   1:L PR[91] R[100]mm/sec CNT100;
   1:  PR[91,1] = PR[90,1] + -28.510;
   1:  PR[91,2] = PR[90,2] + -18.557;
   1:L PR[91] R[100]mm/sec CNT100;
   1:  PR[91,1] = PR[90,1] + -27.839;
   1:  PR[91,2] = PR[90,2] + -18.919;
   1:  PR[91,3] = PR[90,3] + 48.630;
   1:L PR[91] R[100]mm/sec CNT100;
   1:  PR[91,1] = PR[90,1] + -24.290;
   1:  PR[91,2] = PR[90,2] + -20.442;
   1:  PR[91,3] = PR[90,3] + 48.632;
   1:L PR[91] R[100]mm/sec CNT100;
   1:  PR[91,1] = PR[90,1] + -22.878;
   1:  PR[91,2] = PR[90,2] + -20.850;
   1:  PR[91,3] = PR[90,3] + 48.644;
   1:L PR[91] R[100]mm/sec CNT100;
   1:  PR[91,1] = PR[90,1] + -19.713;
   1:  PR[91,2] = PR[90,2] + -21.485;
   1:  PR[91,3] = PR[90,3] + 48.648;
   1:L PR[91] R[100]mm/sec CNT100;
   1:  PR[91,1] = PR[90,1] + -17.392;
   1:  PR[91,2] = PR[90,2] + -21.649;
   1:  PR[91,3] = PR[90,3] + 48.658;
   1:L PR[91] R[100]mm/sec CNT100;
   1:  PR[91,1] = PR[90,1] + -14.946;
   1:  PR[91,2] = PR[90,2] + -21.626;
   1:  PR[91,3] = PR[90,3] + 48.665;
   1:L PR[91] R[100]mm/sec CNT100;
   1:  PR[91,1] = PR[90,1] + -11.689;
   1:  PR[91,2] = PR[90,2] + -21.159;
   1:  PR[91,3] = PR[90,3] + 48.672;
   1:L PR[91] R[100]mm/sec CNT100;
   1:  PR[91,1] = PR[90,1] + -10.176;
   1:  PR[91,2] = PR[90,2] + -20.823;
   1:  PR[91,3] = PR[90,3] + 48.682;
   1:L PR[91] R[100]mm/sec CNT100;
   1:  PR[91,1] = PR[90,1] + -6.157;
   1:  PR[91,2] = PR[90,2] + -19.311;
   1:  PR[91,3] = PR[90,3] + 48.687;
   1:L PR[91] R[100]mm/sec CNT100;
   1:  PR[91,1] = PR[90,1] + -5.614;
   1:  PR[91,2] = PR[90,2] + -19.060;
   1:  PR[91,3] = PR[90,3] + 48.700;
   1:L PR[91] R[100]mm/sec CNT100;
   1:  PR[91,1] = PR[90,1] + -1.632;
   1:  PR[91,2] = PR[90,2] + -16.429;
   1:  PR[91,3] = PR[90,3] + 48.702;
   1:L PR[91] R[100]mm/sec CNT100;
   1:  PR[91,1] = PR[90,1] + -1.354;
   1:  PR[91,2] = PR[90,2] + -16.258;
   1:  PR[91,3] = PR[90,3] + 48.716;
   1:L PR[91] R[100]mm/sec CNT100;
   1:  PR[91,1] = PR[90,1] + 6.289;
   1:  PR[91,2] = PR[90,2] + -8.641;
   1:  PR[91,3] = PR[90,3] + 48.717;
   1:L PR[91] R[100]mm/sec CNT100;
   1:  PR[91,1] = PR[90,1] + 5.337;
   1:  PR[91,2] = PR[90,2] + -14.022;
   1:  PR[91,3] = PR[90,3] + 48.750;
   1:L PR[91] R[100]mm/sec CNT100;
   1:  PR[91,1] = PR[90,1] + 8.828;
   1:  PR[91,2] = PR[90,2] + -17.700;
   1:  PR[91,3] = PR[90,3] + 48.767;
   1:L PR[91] R[100]mm/sec CNT100;
   1:  PR[91,1] = PR[90,1] + 9.012;
   1:  PR[91,2] = PR[90,2] + -17.839;
   1:  PR[91,3] = PR[90,3] + 48.782;
   1:L PR[91] R[100]mm/sec CNT100;
   1:  PR[91,1] = PR[90,1] + 13.464;
   1:  PR[91,2] = PR[90,2] + -20.615;
   1:  PR[91,3] = PR[90,3] + 48.783;
   1:L PR[91] R[100]mm/sec CNT100;
   1:  PR[91,1] = PR[90,1] + 13.849;
   1:  PR[91,2] = PR[90,2] + -20.772;
   1:  PR[91,3] = PR[90,3] + 48.799;
   1:L PR[91] R[100]mm/sec CNT100;
   1:  PR[91,1] = PR[90,1] + 18.670;
   1:  PR[91,2] = PR[90,2] + -22.298;
   1:  PR[91,3] = PR[90,3] + 48.800;
   1:L PR[91] R[100]mm/sec CNT100;
   1:  PR[91,1] = PR[90,1] + 19.283;
   1:  PR[91,2] = PR[90,2] + -22.377;
   1:  PR[91,3] = PR[90,3] + 48.815;
   1:L PR[91] R[100]mm/sec CNT100;
   1:  PR[91,1] = PR[90,1] + 24.125;
   1:  PR[91,2] = PR[90,2] + -22.656;
   1:  PR[91,3] = PR[90,3] + 48.817;
   1:L PR[91] R[100]mm/sec CNT100;
   1:  PR[91,1] = PR[90,1] + 24.941;
   1:  PR[91,2] = PR[90,2] + -22.547;
   1:  PR[91,3] = PR[90,3] + 48.832;
   1:L PR[91] R[100]mm/sec CNT100;
   1:  PR[91,1] = PR[90,1] + 29.498;
   1:  PR[91,2] = PR[90,2] + -21.664;
   1:  PR[91,3] = PR[90,3] + 48.834;
   1:L PR[91] R[100]mm/sec CNT100;
   1:  PR[91,1] = PR[90,1] + 30.441;
   1:  PR[91,2] = PR[90,2] + -21.275;
   1:  PR[91,3] = PR[90,3] + 48.848;
   1:L PR[91] R[100]mm/sec CNT100;
   1:  PR[91,1] = PR[90,1] + 34.460;
   1:  PR[91,2] = PR[90,2] + -19.387;
   1:  PR[91,3] = PR[90,3] + 48.852;
   1:L PR[91] R[100]mm/sec CNT100;
   1:  PR[91,1] = PR[90,1] + 35.553;
   1:  PR[91,2] = PR[90,2] + -18.557;
   1:  PR[91,3] = PR[90,3] + 48.865;
   1:L PR[91] R[100]mm/sec CNT100;
   1:  PR[91,1] = PR[90,1] + 35.978;
   1:  PR[91,2] = PR[90,2] + -18.324;
   1:  PR[91,3] = PR[90,3] + 48.869;
   1:L PR[91] R[100]mm/sec CNT100;
   1:  PR[91,1] = PR[90,1] + 37.531;
   1:  PR[91,2] = PR[90,2] + -17.267;
   1:  PR[91,3] = PR[90,3] + 48.871;
   1:L PR[91] R[100]mm/sec CNT100;
   1:  PR[91,1] = PR[90,1] + 42.420;
   1:  PR[91,2] = PR[90,2] + -19.709;
   1:  PR[91,3] = PR[90,3] + 48.876;
   1:L PR[91] R[100]mm/sec CNT100;
   1:  PR[91,1] = PR[90,1] + 47.455;
   1:  PR[91,2] = PR[90,2] + -21.552;
   1:  PR[91,3] = PR[90,3] + 48.893;
   1:L PR[91] R[100]mm/sec CNT100;
   1:  PR[91,1] = PR[90,1] + 47.820;
   1:  PR[91,2] = PR[90,2] + -21.671;
   1:  PR[91,3] = PR[90,3] + 48.909;
   1:L PR[91] R[100]mm/sec CNT100;
   1:  PR[91,1] = PR[90,1] + 48.269;
   1:  PR[91,2] = PR[90,2] + -21.751;
   1:  PR[91,3] = PR[90,3] + 48.910;
   1:L PR[91] R[100]mm/sec CNT100;
   1:  PR[91,1] = PR[90,1] + 52.654;
   1:  PR[91,2] = PR[90,2] + -22.644;
   1:  PR[91,3] = PR[90,3] + 48.912;
   1:L PR[91] R[100]mm/sec CNT100;
   1:  PR[91,1] = PR[90,1] + 55.223;
   1:  PR[91,2] = PR[90,2] + -23.107;
   1:  PR[91,3] = PR[90,3] + 48.925;
   1:L PR[91] R[100]mm/sec CNT100;
   1:  PR[91,1] = PR[90,1] + 57.159;
   1:  PR[91,2] = PR[90,2] + -23.143;
   1:  PR[91,3] = PR[90,3] + 48.933;
   1:L PR[91] R[100]mm/sec CNT100;
   1:  PR[91,1] = PR[90,1] + 61.173;
   1:  PR[91,2] = PR[90,2] + -23.148;
   1:  PR[91,3] = PR[90,3] + 48.939;
   1:L PR[91] R[100]mm/sec CNT100;
   1:  PR[91,1] = PR[90,1] + 62.107;
   1:  PR[91,2] = PR[90,2] + -23.164;
   1:  PR[91,3] = PR[90,3] + 48.951;
   1:L PR[91] R[100]mm/sec CNT100;
   1:  PR[91,1] = PR[90,1] + 62.457;
   1:  PR[91,2] = PR[90,2] + -23.132;
   1:  PR[91,3] = PR[90,3] + 48.954;
   1:L PR[91] R[100]mm/sec CNT100;
   1:  PR[91,1] = PR[90,1] + 67.159;
   1:  PR[91,2] = PR[90,2] + -22.316;
   1:  PR[91,3] = PR[90,3] + 48.955;
   1:L PR[91] R[100]mm/sec CNT100;
   1:  PR[91,1] = PR[90,1] + 69.950;
   1:  PR[91,2] = PR[90,2] + -21.478;
   1:  PR[91,3] = PR[90,3] + 48.970;
   1:L PR[91] R[100]mm/sec CNT100;
   1:  PR[91,1] = PR[90,1] + 72.162;
   1:  PR[91,2] = PR[90,2] + -20.641;
   1:  PR[91,3] = PR[90,3] + 48.979;
   1:L PR[91] R[100]mm/sec CNT100;
   1:  PR[91,1] = PR[90,1] + 76.463;
   1:  PR[91,2] = PR[90,2] + -18.303;
   1:  PR[91,3] = PR[90,3] + 48.986;
   1:L PR[91] R[100]mm/sec CNT100;
   1:  PR[91,1] = PR[90,1] + 76.838;
   1:  PR[91,2] = PR[90,2] + -18.068;
   1:  PR[91,3] = PR[90,3] + 49.001;
   1:L PR[91] R[100]mm/sec CNT100;
   1:  PR[91,1] = PR[90,1] + 78.701;
   1:  PR[91,2] = PR[90,2] + -16.455;
   1:  PR[91,3] = PR[90,3] + 49.002;
   1:L PR[91] R[100]mm/sec CNT100;
   1:  PR[91,1] = PR[90,1] + 80.712;
   1:  PR[91,2] = PR[90,2] + -14.659;
   1:  PR[91,3] = PR[90,3] + 49.009;
   1:L PR[91] R[100]mm/sec CNT100;
   1:  PR[91,1] = PR[90,1] + 80.884;
   1:  PR[91,2] = PR[90,2] + -14.488;
   1:  PR[91,3] = PR[90,3] + 49.018;
   1:L PR[91] R[100]mm/sec CNT100;
   1:  PR[91,1] = PR[90,1] + 83.396;
   1:  PR[91,2] = PR[90,2] + -10.888;
   1:L PR[91] R[100]mm/sec CNT100;
   1:  PR[91,1] = PR[90,1] + 83.851;
   1:  PR[91,2] = PR[90,2] + -10.181;
   1:  PR[91,3] = PR[90,3] + 49.032;
   1:L PR[91] R[100]mm/sec CNT100;
   1:  PR[91,1] = PR[90,1] + 85.213;
   1:  PR[91,2] = PR[90,2] + -6.661;
   1:  PR[91,3] = PR[90,3] + 49.034;
   1:L PR[91] R[100]mm/sec CNT100;
   1:  PR[91,1] = PR[90,1] + 85.617;
   1:  PR[91,2] = PR[90,2] + -5.543;
   1:  PR[91,3] = PR[90,3] + 49.046;
   1:L PR[91] R[100]mm/sec CNT100;
   1:  PR[91,1] = PR[90,1] + 85.782;
   1:  PR[91,2] = PR[90,2] + -4.149;
   1:  PR[91,3] = PR[90,3] + 49.049;
   1:L PR[91] R[100]mm/sec CNT100;
   1:  PR[91,1] = PR[90,1] + 85.832;
   1:  PR[91,2] = PR[90,2] + -3.920;
   1:  PR[91,3] = PR[90,3] + 49.053;
   1:L PR[91] R[100]mm/sec CNT100;
   1:  PR[91,1] = PR[90,1] + 86.226;
   1:  PR[91,2] = PR[90,2] + -0.738;
   1:  PR[91,3] = PR[90,3] + 49.054;
   1:L PR[91] R[100]mm/sec CNT100;
   1:  PR[91,1] = PR[90,1] + 86.045;
   1:  PR[91,2] = PR[90,2] + 0.626;
   1:  PR[91,3] = PR[90,3] + 49.064;
   1:L PR[91] R[100]mm/sec CNT100;
   1:  PR[91,1] = PR[90,1] + 85.619;
   1:  PR[91,2] = PR[90,2] + 4.079;
   1:  PR[91,3] = PR[90,3] + 49.068;
   1:L PR[91] R[100]mm/sec CNT100;
   1:  PR[91,1] = PR[90,1] + 85.213;
   1:  PR[91,2] = PR[90,2] + 5.202;
   1:  PR[91,3] = PR[90,3] + 49.079;
   1:L PR[91] R[100]mm/sec CNT100;
   1:  PR[91,1] = PR[90,1] + 83.852;
   1:  PR[91,2] = PR[90,2] + 8.722;
   1:  PR[91,3] = PR[90,3] + 49.082;
   1:L PR[91] R[100]mm/sec CNT100;
   1:  PR[91,1] = PR[90,1] + 83.396;
   1:  PR[91,2] = PR[90,2] + 9.429;
   1:  PR[91,3] = PR[90,3] + 49.094;
   1:L PR[91] R[100]mm/sec CNT100;
   1:  PR[91,1] = PR[90,1] + 80.884;
   1:  PR[91,2] = PR[90,2] + 13.029;
   1:  PR[91,3] = PR[90,3] + 49.096;
   1:L PR[91] R[100]mm/sec CNT100;
   1:  PR[91,1] = PR[90,1] + 80.712;
   1:  PR[91,2] = PR[90,2] + 13.200;
   1:  PR[91,3] = PR[90,3] + 49.110;
   1:L PR[91] R[100]mm/sec CNT100;
   1:  PR[91,1] = PR[90,1] + 78.702;
   1:  PR[91,2] = PR[90,2] + 14.996;
   1:L PR[91] R[100]mm/sec CNT100;
   1:  PR[91,1] = PR[90,1] + 76.837;
   1:  PR[91,2] = PR[90,2] + 16.610;
   1:  PR[91,3] = PR[90,3] + 49.118;
   1:L PR[91] R[100]mm/sec CNT100;
   1:  PR[91,1] = PR[90,1] + 76.458;
   1:  PR[91,2] = PR[90,2] + 16.846;
   1:  PR[91,3] = PR[90,3] + 49.126;
   1:L PR[91] R[100]mm/sec CNT100;
   1:  PR[91,1] = PR[90,1] + 72.151;
   1:  PR[91,2] = PR[90,2] + 19.188;
   1:  PR[91,3] = PR[90,3] + 49.127;
   1:L PR[91] R[100]mm/sec CNT100;
   1:  PR[91,1] = PR[90,1] + 69.917;
   1:  PR[91,2] = PR[90,2] + 20.029;
   1:  PR[91,3] = PR[90,3] + 49.142;
   1:L PR[91] R[100]mm/sec CNT100;
   1:  PR[91,1] = PR[90,1] + 67.130;
   1:  PR[91,2] = PR[90,2] + 20.866;
   1:  PR[91,3] = PR[90,3] + 49.149;
   1:L PR[91] R[100]mm/sec CNT100;
   1:  PR[91,1] = PR[90,1] + 62.374;
   1:  PR[91,2] = PR[90,2] + 21.681;
   1:  PR[91,3] = PR[90,3] + 49.158;
   1:L PR[91] R[100]mm/sec CNT100;
   1:  PR[91,1] = PR[90,1] + 62.052;
   1:  PR[91,2] = PR[90,2] + 21.710;
   1:  PR[91,3] = PR[90,3] + 49.173;
   1:L PR[91] R[100]mm/sec CNT100;
   1:  PR[91,1] = PR[90,1] + 61.178;
   1:  PR[91,2] = PR[90,2] + 21.693;
   1:  PR[91,3] = PR[90,3] + 49.174;
   1:L PR[91] R[100]mm/sec CNT100;
   1:  PR[91,1] = PR[90,1] + 57.119;
   1:  PR[91,2] = PR[90,2] + 21.677;
   1:  PR[91,3] = PR[90,3] + 49.176;
   1:L PR[91] R[100]mm/sec CNT100;
   1:  PR[91,1] = PR[90,1] + 55.187;
   1:  PR[91,2] = PR[90,2] + 21.645;
   1:  PR[91,3] = PR[90,3] + 49.189;
   1:L PR[91] R[100]mm/sec CNT100;
   1:  PR[91,1] = PR[90,1] + 52.645;
   1:  PR[91,2] = PR[90,2] + 21.178;
   1:  PR[91,3] = PR[90,3] + 49.195;
   1:L PR[91] R[100]mm/sec CNT100;
   1:  PR[91,1] = PR[90,1] + 48.267;
   1:  PR[91,2] = PR[90,2] + 20.296;
   1:  PR[91,3] = PR[90,3] + 49.202;
   1:L PR[91] R[100]mm/sec CNT100;
   1:  PR[91,1] = PR[90,1] + 47.858;
   1:  PR[91,2] = PR[90,2] + 20.223;
   1:  PR[91,3] = PR[90,3] + 49.216;
   1:L PR[91] R[100]mm/sec CNT100;
   1:  PR[91,1] = PR[90,1] + 47.525;
   1:  PR[91,2] = PR[90,2] + 20.114;
   1:  PR[91,3] = PR[90,3] + 49.217;
   1:L PR[91] R[100]mm/sec CNT100;
   1:  PR[91,1] = PR[90,1] + 42.433;
   1:  PR[91,2] = PR[90,2] + 18.257;
   1:  PR[91,3] = PR[90,3] + 49.218;
   1:L PR[91] R[100]mm/sec CNT100;
   1:  PR[91,1] = PR[90,1] + 37.498;
   1:  PR[91,2] = PR[90,2] + 15.791;
   1:  PR[91,3] = PR[90,3] + 49.235;
   1:L PR[91] R[100]mm/sec CNT100;
   1:  PR[91,1] = PR[90,1] + 35.153;
   1:  PR[91,2] = PR[90,2] + 17.482;
   1:  PR[91,3] = PR[90,3] + 49.252;
   1:L PR[91] R[100]mm/sec CNT100;
   1:  PR[91,1] = PR[90,1] + 34.510;
   1:  PR[91,2] = PR[90,2] + 17.906;
   1:  PR[91,3] = PR[90,3] + 49.260;
   1:L PR[91] R[100]mm/sec CNT100;
   1:  PR[91,1] = PR[90,1] + 30.435;
   1:  PR[91,2] = PR[90,2] + 19.820;
   1:  PR[91,3] = PR[90,3] + 49.263;
   1:L PR[91] R[100]mm/sec CNT100;
   1:  PR[91,1] = PR[90,1] + 29.493;
   1:  PR[91,2] = PR[90,2] + 20.206;
   1:  PR[91,3] = PR[90,3] + 49.276;
   1:L PR[91] R[100]mm/sec CNT100;
   1:  PR[91,1] = PR[90,1] + 24.940;
   1:  PR[91,2] = PR[90,2] + 21.089;
   1:  PR[91,3] = PR[90,3] + 49.279;
   1:L PR[91] R[100]mm/sec CNT100;
   1:  PR[91,1] = PR[90,1] + 24.124;
   1:  PR[91,2] = PR[90,2] + 21.197;
   1:  PR[91,3] = PR[90,3] + 49.293;
   1:L PR[91] R[100]mm/sec CNT100;
   1:  PR[91,1] = PR[90,1] + 19.286;
   1:  PR[91,2] = PR[90,2] + 20.919;
   1:  PR[91,3] = PR[90,3] + 49.296;
   1:L PR[91] R[100]mm/sec CNT100;
   1:  PR[91,1] = PR[90,1] + 18.673;
   1:  PR[91,2] = PR[90,2] + 20.840;
   1:  PR[91,3] = PR[90,3] + 49.311;
   1:L PR[91] R[100]mm/sec CNT100;
   1:  PR[91,1] = PR[90,1] + 13.856;
   1:  PR[91,2] = PR[90,2] + 19.317;
   1:  PR[91,3] = PR[90,3] + 49.313;
   1:L PR[91] R[100]mm/sec CNT100;
   1:  PR[91,1] = PR[90,1] + 13.471;
   1:  PR[91,2] = PR[90,2] + 19.160;
   1:  PR[91,3] = PR[90,3] + 49.328;
   1:L PR[91] R[100]mm/sec CNT100;
   1:  PR[91,1] = PR[90,1] + 9.021;
   1:  PR[91,2] = PR[90,2] + 16.388;
   1:  PR[91,3] = PR[90,3] + 49.329;
   1:L PR[91] R[100]mm/sec CNT100;
   1:  PR[91,1] = PR[90,1] + 8.837;
   1:  PR[91,2] = PR[90,2] + 16.249;
   1:  PR[91,3] = PR[90,3] + 49.345;
   1:L PR[91] R[100]mm/sec CNT100;
   1:  PR[91,1] = PR[90,1] + 5.077;
   1:  PR[91,2] = PR[90,2] + 12.292;
   1:  PR[91,3] = PR[90,3] + 49.346;
   1:L PR[91] R[100]mm/sec CNT100;
   1:  PR[91,1] = PR[90,1] + 3.469;
   1:  PR[91,2] = PR[90,2] + 10.055;
   1:  PR[91,3] = PR[90,3] + 49.362;
   1:L PR[91] R[100]mm/sec CNT100;
   1:  PR[91,1] = PR[90,1] + -1.325;
   1:  PR[91,2] = PR[90,2] + 14.778;
   1:  PR[91,3] = PR[90,3] + 49.371;
   1:L PR[91] R[100]mm/sec CNT100;
   1:  PR[91,1] = PR[90,1] + -1.634;
   1:  PR[91,2] = PR[90,2] + 14.968;
   1:  PR[91,3] = PR[90,3] + 49.391;
   1:L PR[91] R[100]mm/sec CNT100;
   1:  PR[91,1] = PR[90,1] + -5.589;
   1:  PR[91,2] = PR[90,2] + 17.588;
   1:  PR[91,3] = PR[90,3] + 49.392;
   1:L PR[91] R[100]mm/sec CNT100;
   1:  PR[91,1] = PR[90,1] + -6.128;
   1:  PR[91,2] = PR[90,2] + 17.838;
   1:  PR[91,3] = PR[90,3] + 49.407;
   1:L PR[91] R[100]mm/sec CNT100;
   1:  PR[91,1] = PR[90,1] + -10.150;
   1:  PR[91,2] = PR[90,2] + 19.357;
   1:  PR[91,3] = PR[90,3] + 49.408;
   1:L PR[91] R[100]mm/sec CNT100;
   1:  PR[91,1] = PR[90,1] + -11.659;
   1:  PR[91,2] = PR[90,2] + 19.694;
   1:  PR[91,3] = PR[90,3] + 49.421;
   1:L PR[91] R[100]mm/sec CNT100;
   1:  PR[91,1] = PR[90,1] + -14.921;
   1:  PR[91,2] = PR[90,2] + 20.165;
   1:  PR[91,3] = PR[90,3] + 49.426;
   1:L PR[91] R[100]mm/sec CNT100;
   1:  PR[91,1] = PR[90,1] + -17.365;
   1:  PR[91,2] = PR[90,2] + 20.190;
   1:  PR[91,3] = PR[90,3] + 49.436;
   1:L PR[91] R[100]mm/sec CNT100;
   1:  PR[91,1] = PR[90,1] + -19.691;
   1:  PR[91,2] = PR[90,2] + 20.030;
   1:  PR[91,3] = PR[90,3] + 49.443;
   1:L PR[91] R[100]mm/sec CNT100;
   1:  PR[91,1] = PR[90,1] + -22.856;
   1:  PR[91,2] = PR[90,2] + 19.396;
   1:  PR[91,3] = PR[90,3] + 49.451;
   1:L PR[91] R[100]mm/sec CNT100;
   1:  PR[91,1] = PR[90,1] + -24.272;
   1:  PR[91,2] = PR[90,2] + 18.990;
   1:  PR[91,3] = PR[90,3] + 49.460;
   1:L PR[91] R[100]mm/sec CNT100;
   1:  PR[91,1] = PR[90,1] + -27.822;
   1:  PR[91,2] = PR[90,2] + 17.468;
   1:  PR[91,3] = PR[90,3] + 49.465;
   1:L PR[91] R[100]mm/sec CNT100;
   1:  PR[91,1] = PR[90,1] + -28.488;
   1:  PR[91,2] = PR[90,2] + 17.112;
   1:  PR[91,3] = PR[90,3] + 49.476;
   1:L PR[91] R[100]mm/sec CNT100;
   1:  PR[91,1] = PR[90,1] + -32.086;
   1:  PR[91,2] = PR[90,2] + 14.574;
   1:  PR[91,3] = PR[90,3] + 49.479;
   1:L PR[91] R[100]mm/sec CNT100;
   1:  PR[91,1] = PR[90,1] + -32.241;
   1:  PR[91,2] = PR[90,2] + 14.449;
   1:  PR[91,3] = PR[90,3] + 49.492;
   1:L PR[91] R[100]mm/sec CNT100;
   1:  PR[91,1] = PR[90,1] + -33.278;
   1:  PR[91,2] = PR[90,2] + 13.352;
   1:  PR[91,3] = PR[90,3] + 49.493;
   1:L PR[91] R[100]mm/sec CNT100;
   1:  PR[91,1] = PR[90,1] + -36.656;
   1:  PR[91,2] = PR[90,2] + 9.566;
   1:  PR[91,3] = PR[90,3] + 49.497;
   1:L PR[91] R[100]mm/sec CNT100;
   1:  PR[91,1] = PR[90,1] + -41.550;
   1:  PR[91,2] = PR[90,2] + 13.514;
   1:  PR[91,3] = PR[90,3] + 49.513;
   1:L PR[91] R[100]mm/sec CNT100;
   1:  PR[91,1] = PR[90,1] + -43.321;
   1:  PR[91,2] = PR[90,2] + 14.828;
   1:  PR[91,3] = PR[90,3] + 49.532;
   1:L PR[91] R[100]mm/sec CNT100;
   1:  PR[91,1] = PR[90,1] + -44.951;
   1:  PR[91,2] = PR[90,2] + 15.641;
   1:  PR[91,3] = PR[90,3] + 49.538;
   1:L PR[91] R[100]mm/sec CNT100;
   1:  PR[91,1] = PR[90,1] + -48.152;
   1:  PR[91,2] = PR[90,2] + 17.124;
   1:  PR[91,3] = PR[90,3] + 49.544;
   1:L PR[91] R[100]mm/sec CNT100;
   1:  PR[91,1] = PR[90,1] + -49.267;
   1:  PR[91,2] = PR[90,2] + 17.701;
   1:  PR[91,3] = PR[90,3] + 49.555;
   1:L PR[91] R[100]mm/sec CNT100;
   1:  PR[91,1] = PR[90,1] + -52.863;
   1:  PR[91,2] = PR[90,2] + 18.796;
   1:  PR[91,3] = PR[90,3] + 49.559;
   1:L PR[91] R[100]mm/sec CNT100;
   1:  PR[91,1] = PR[90,1] + -55.102;
   1:  PR[91,2] = PR[90,2] + 19.415;
   1:  PR[91,3] = PR[90,3] + 49.570;
   1:L PR[91] R[100]mm/sec CNT100;
   1:  PR[91,1] = PR[90,1] + -56.835;
   1:  PR[91,2] = PR[90,2] + 19.617;
   1:  PR[91,3] = PR[90,3] + 49.577;
   1:L PR[91] R[100]mm/sec CNT100;
   1:  PR[91,1] = PR[90,1] + -61.020;
   1:  PR[91,2] = PR[90,2] + 20.022;
   1:  PR[91,3] = PR[90,3] + 49.582;
   1:L PR[91] R[100]mm/sec CNT100;
   1:  PR[91] = PR[90];
   1:  PR[91,1] = PR[90,1] + -65.410;
   1:  PR[91,2] = PR[90,2] + 19.840;
   1:  PR[91,3] = PR[90,3] + 50.895;
   1:L PR[91] R[100]mm/sec CNT100;
   1:  PR[91,1] = PR[90,1] + -70.231;
   1:  PR[91,2] = PR[90,2] + 18.648;
   1:  PR[91,3] = PR[90,3] + 49.612;
   1:L PR[91] R[100]mm/sec CNT100;
   1:  PR[91,1] = PR[90,1] + -72.512;
   1:  PR[91,2] = PR[90,2] + 17.632;
   1:  PR[91,3] = PR[90,3] + 49.627;
   1:L PR[91] R[100]mm/sec CNT100;
   1:  PR[91,1] = PR[90,1] + -74.603;
   1:  PR[91,2] = PR[90,2] + 16.680;
   1:  PR[91,3] = PR[90,3] + 49.635;
   1:L PR[91] R[100]mm/sec CNT100;
   1:  PR[91,1] = PR[90,1] + -77.632;
   1:  PR[91,2] = PR[90,2] + 14.570;
   1:  PR[91,3] = PR[90,3] + 49.642;
   1:L PR[91] R[100]mm/sec CNT100;
   1:  PR[91,1] = PR[90,1] + -78.386;
   1:  PR[91,2] = PR[90,2] + 14.036;
   1:  PR[91,3] = PR[90,3] + 49.653;
   1:L PR[91] R[100]mm/sec CNT100;
   1:  PR[91,1] = PR[90,1] + -81.455;
   1:  PR[91,2] = PR[90,2] + 10.830;
   1:  PR[91,3] = PR[90,3] + 49.656;
   1:L PR[91] R[100]mm/sec CNT100;
   1:  PR[91,1] = PR[90,1] + -82.214;
   1:  PR[91,2] = PR[90,2] + 9.609;
   1:  PR[91,3] = PR[90,3] + 49.670;
   1:L PR[91] R[100]mm/sec CNT100;
   1:  PR[91,1] = PR[90,1] + -83.620;
   1:  PR[91,2] = PR[90,2] + 7.244;
   1:  PR[91,3] = PR[90,3] + 49.674;
   1:L PR[91] R[100]mm/sec CNT100;
   1:  PR[91,1] = PR[90,1] + -84.935;
   1:  PR[91,2] = PR[90,2] + 3.331;
   1:  PR[91,3] = PR[90,3] + 49.683;
   1:L PR[91] R[100]mm/sec CNT100;
   1:  PR[91,1] = PR[90,1] + -84.977;
   1:  PR[91,2] = PR[90,2] + 2.953;
   1:  PR[91,3] = PR[90,3] + 49.695;
   1:L PR[91] R[100]mm/sec CNT100;
   1:  PR[91,1] = PR[90,1] + -85.030;
   1:  PR[91,2] = PR[90,2] + 2.675;
   1:  PR[91,3] = PR[90,3] + 49.696;
   1:L PR[91] R[100]mm/sec CNT100;
   1:  PR[91,1] = PR[90,1] + -85.403;
   1:  PR[91,2] = PR[90,2] + -0.728;
   1:  PR[91,3] = PR[90,3] + 49.697;
   1:L PR[91] R[100]mm/sec CNT100;
   1:  PR[91,1] = PR[90,1] + -85.339;
   1:  PR[91,2] = PR[90,2] + -1.306;
   1:  PR[91,3] = PR[90,3] + 49.708;
   1:L PR[91] R[100]mm/sec CNT100;
   1:  PR[91,1] = PR[90,1] + -85.045;
   1:  PR[91,2] = PR[90,2] + -2.662;
   1:  PR[91,3] = PR[90,3] + 49.710;
   1:L PR[91] R[100]mm/sec CNT100;
   1:  PR[91,1] = PR[90,1] + -84.811;
   1:  PR[91,2] = PR[90,2] + -4.786;
   1:  PR[91,3] = PR[90,3] + 49.714;
   1:L PR[91] R[100]mm/sec CNT100;
   1:  PR[91,1] = PR[90,1] + -84.183;
   1:  PR[91,2] = PR[90,2] + -6.613;
   1:  PR[91,3] = PR[90,3] + 49.720;
   1:L PR[91] R[100]mm/sec CNT100;
   1:  PR[91,1] = PR[90,1] + -83.474;
   1:  PR[91,2] = PR[90,2] + -8.702;
   1:  PR[91,3] = PR[90,3] + 49.726;
   1:L PR[91] R[100]mm/sec CNT100;
   1:  PR[91,1] = PR[90,1] + -81.289;
   1:  PR[91,2] = PR[90,2] + -12.323;
   1:  PR[91,3] = PR[90,3] + 49.733;
   1:L PR[91] R[100]mm/sec CNT100;
   1:  PR[91,1] = PR[90,1] + -78.321;
   1:  PR[91,2] = PR[90,2] + -15.514;
   1:  PR[91,3] = PR[90,3] + 49.746;
   1:L PR[91] R[100]mm/sec CNT100;
   1:  PR[91,1] = PR[90,1] + -74.667;
   1:  PR[91,2] = PR[90,2] + -18.139;
   1:  PR[91,3] = PR[90,3] + 49.760;
   1:L PR[91] R[100]mm/sec CNT100;
   1:  PR[91,1] = PR[90,1] + -72.890;
   1:  PR[91,2] = PR[90,2] + -18.954;
   1:  PR[91,3] = PR[90,3] + 49.773;
   1:L PR[91] R[100]mm/sec CNT100;
   1:  PR[91,1] = PR[90,1] + -70.561;
   1:  PR[91,2] = PR[90,2] + -19.988;
   1:  PR[91,3] = PR[90,3] + 49.779;
   1:L PR[91] R[100]mm/sec CNT100;
   1:  PR[91,1] = PR[90,1] + -70.100;
   1:  PR[91,2] = PR[90,2] + -20.163;
   1:  PR[91,3] = PR[90,3] + 49.787;
   1:L PR[91] R[100]mm/sec CNT100;
   1:  PR[91,1] = PR[90,1] + -66.353;
   1:  PR[91,2] = PR[90,2] + -21.081;
   1:  PR[91,3] = PR[90,3] + 49.789;
   1:L PR[91] R[100]mm/sec CNT100;
   1:  PR[91,1] = PR[90,1] + -64.382;
   1:  PR[91,2] = PR[90,2] + -21.432;
   1:  PR[91,3] = PR[90,3] + 49.801;
   1:L PR[91] R[100]mm/sec CNT100;
   1:  PR[91,1] = PR[90,1] + -61.899;
   1:  PR[91,2] = PR[90,2] + -21.598;
   1:  PR[91,3] = PR[90,3] + 49.807;
   1:L PR[91] R[100]mm/sec CNT100;
   1:  PR[91,1] = PR[90,1] + -57.979;
   1:  PR[91,2] = PR[90,2] + -21.564;
   1:  PR[91,3] = PR[90,3] + 49.814;
   1:L PR[91] R[100]mm/sec CNT100;
   1:  PR[91,1] = PR[90,1] + -57.272;
   1:  PR[91,2] = PR[90,2] + -21.487;
   1:  PR[91,3] = PR[90,3] + 49.826;
   1:L PR[91] R[100]mm/sec CNT100;
   1:  PR[91,1] = PR[90,1] + -55.108;
   1:  PR[91,2] = PR[90,2] + -21.058;
   1:  PR[91,3] = PR[90,3] + 49.829;
   1:L PR[91] R[100]mm/sec CNT100;
   1:  PR[91,1] = PR[90,1] + -51.613;
   1:  PR[91,2] = PR[90,2] + -20.501;
   1:  PR[91,3] = PR[90,3] + 49.835;
   1:L PR[91] R[100]mm/sec CNT100;
   1:  PR[91,1] = PR[90,1] + -48.807;
   1:  PR[91,2] = PR[90,2] + -19.545;
   1:  PR[91,3] = PR[90,3] + 49.846;
   1:L PR[91] R[100]mm/sec CNT100;
   1:  PR[91,1] = PR[90,1] + -45.807;
   1:  PR[91,2] = PR[90,2] + -18.487;
   1:  PR[91,3] = PR[90,3] + 49.855;
   1:L PR[91] R[100]mm/sec CNT100;
   1:  PR[91,1] = PR[90,1] + -42.369;
   1:  PR[91,2] = PR[90,2] + -16.486;
   1:  PR[91,3] = PR[90,3] + 49.865;
   1:L PR[91] R[100]mm/sec CNT100;
   1:  PR[91,1] = PR[90,1] + -40.708;
   1:  PR[91,2] = PR[90,2] + -15.676;
   1:  PR[91,3] = PR[90,3] + 49.877;
   1:L PR[91] R[100]mm/sec CNT100;
   1:  PR[91,1] = PR[90,1] + -39.853;
   1:  PR[91,2] = PR[90,2] + -15.176;
   1:  PR[91,3] = PR[90,3] + 49.883;
   1:L PR[91] R[100]mm/sec CNT100;
   1:  PR[91,1] = PR[90,1] + -35.756;
   1:  PR[91,2] = PR[90,2] + -11.923;
   1:  PR[91,3] = PR[90,3] + 49.886;
   1:L PR[91] R[100]mm/sec CNT100;
   1:  PR[91,1] = PR[90,1] + -32.347;
   1:  PR[91,2] = PR[90,2] + -15.600;
   1:  PR[91,3] = PR[90,3] + 49.902;
   1:L PR[91] R[100]mm/sec CNT100;
   1:  PR[91,1] = PR[90,1] + -32.174;
   1:  PR[91,2] = PR[90,2] + -15.768;
   1:  PR[91,3] = PR[90,3] + 49.918;
   1:L PR[91] R[100]mm/sec CNT100;
   1:  PR[91,1] = PR[90,1] + -31.539;
   1:  PR[91,2] = PR[90,2] + -16.296;
   1:L PR[91] R[100]mm/sec CNT100;
   1:  PR[91,1] = PR[90,1] + -28.313;
   1:  PR[91,2] = PR[90,2] + -18.567;
   1:  PR[91,3] = PR[90,3] + 49.921;
   1:L PR[91] R[100]mm/sec CNT100;
   1:  PR[91,1] = PR[90,1] + -27.108;
   1:  PR[91,2] = PR[90,2] + -19.217;
   1:  PR[91,3] = PR[90,3] + 49.933;
   1:L PR[91] R[100]mm/sec CNT100;
   1:  PR[91,1] = PR[90,1] + -24.076;
   1:  PR[91,2] = PR[90,2] + -20.518;
   1:  PR[91,3] = PR[90,3] + 49.937;
   1:L PR[91] R[100]mm/sec CNT100;
   1:  PR[91,1] = PR[90,1] + -22.050;
   1:  PR[91,2] = PR[90,2] + -21.103;
   1:  PR[91,3] = PR[90,3] + 49.947;
   1:L PR[91] R[100]mm/sec CNT100;
   1:  PR[91,1] = PR[90,1] + -19.474;
   1:  PR[91,2] = PR[90,2] + -21.621;
   1:  PR[91,3] = PR[90,3] + 49.954;
   1:L PR[91] R[100]mm/sec CNT100;
   1:  PR[91,1] = PR[90,1] + -16.471;
   1:  PR[91,2] = PR[90,2] + -21.832;
   1:  PR[91,3] = PR[90,3] + 49.962;
   1:L PR[91] R[100]mm/sec CNT100;
   1:  PR[91,1] = PR[90,1] + -14.666;
   1:  PR[91,2] = PR[90,2] + -21.815;
   1:  PR[91,3] = PR[90,3] + 49.971;
   1:L PR[91] R[100]mm/sec CNT100;
   1:  PR[91,1] = PR[90,1] + -10.689;
   1:  PR[91,2] = PR[90,2] + -21.245;
   1:  PR[91,3] = PR[90,3] + 49.977;
   1:L PR[91] R[100]mm/sec CNT100;
   1:  PR[91,1] = PR[90,1] + -9.844;
   1:  PR[91,2] = PR[90,2] + -21.057;
   1:  PR[91,3] = PR[90,3] + 49.989;
   1:L PR[91] R[100]mm/sec CNT100;
   1:  PR[91,1] = PR[90,1] + -5.151;
   1:  PR[91,2] = PR[90,2] + -19.285;
   1:  PR[91,3] = PR[90,3] + 49.992;
   1:L PR[91] R[100]mm/sec CNT100;
   1:  PR[91,1] = PR[90,1] + -4.792;
   1:  PR[91,2] = PR[90,2] + -19.047;
   1:  PR[91,3] = PR[90,3] + 50.007;
   1:L PR[91] R[100]mm/sec CNT100;
   1:  PR[91,1] = PR[90,1] + -0.613;
   1:  PR[91,2] = PR[90,2] + -16.483;
   1:  PR[91,3] = PR[90,3] + 50.008;
   1:L PR[91] R[100]mm/sec CNT100;
   1:  PR[91,1] = PR[90,1] + 0.062;
   1:  PR[91,2] = PR[90,2] + -15.857;
   1:  PR[91,3] = PR[90,3] + 50.023;
   1:L PR[91] R[100]mm/sec CNT100;
   1:  PR[91,1] = PR[90,1] + 6.499;
   1:  PR[91,2] = PR[90,2] + -9.430;
   1:  PR[91,3] = PR[90,3] + 50.026;
   1:L PR[91] R[100]mm/sec CNT100;
   1:  PR[91,1] = PR[90,1] + 5.565;
   1:  PR[91,2] = PR[90,2] + -14.714;
   1:  PR[91,3] = PR[90,3] + 50.054;
   1:L PR[91] R[100]mm/sec CNT100;
   1:  PR[91,1] = PR[90,1] + 8.593;
   1:  PR[91,2] = PR[90,2] + -17.848;
   1:  PR[91,3] = PR[90,3] + 50.071;
   1:L PR[91] R[100]mm/sec CNT100;
   1:  PR[91,1] = PR[90,1] + 8.638;
   1:  PR[91,2] = PR[90,2] + -17.891;
   1:  PR[91,3] = PR[90,3] + 50.084;
   1:L PR[91] R[100]mm/sec CNT100;
   1:  PR[91,1] = PR[90,1] + 13.397;
   1:  PR[91,2] = PR[90,2] + -20.851;
   1:L PR[91] R[100]mm/sec CNT100;
   1:  PR[91,1] = PR[90,1] + 18.676;
   1:  PR[91,2] = PR[90,2] + -22.522;
   1:  PR[91,3] = PR[90,3] + 50.101;
   1:L PR[91] R[100]mm/sec CNT100;
   1:  PR[91,1] = PR[90,1] + 18.762;
   1:  PR[91,2] = PR[90,2] + -22.533;
   1:  PR[91,3] = PR[90,3] + 50.118;
   1:L PR[91] R[100]mm/sec CNT100;
   1:  PR[91,1] = PR[90,1] + 24.160;
   1:  PR[91,2] = PR[90,2] + -22.844;
   1:  PR[91,3] = PR[90,3] + 50.119;
   1:L PR[91] R[100]mm/sec CNT100;
   1:  PR[91,1] = PR[90,1] + 24.456;
   1:  PR[91,2] = PR[90,2] + -22.804;
   1:  PR[91,3] = PR[90,3] + 50.135;
   1:L PR[91] R[100]mm/sec CNT100;
   1:  PR[91,1] = PR[90,1] + 29.553;
   1:  PR[91,2] = PR[90,2] + -21.817;
   1:  PR[91,3] = PR[90,3] + 50.136;
   1:L PR[91] R[100]mm/sec CNT100;
   1:  PR[91,1] = PR[90,1] + 30.017;
   1:  PR[91,2] = PR[90,2] + -21.625;
   1:  PR[91,3] = PR[90,3] + 50.152;
   1:L PR[91] R[100]mm/sec CNT100;
   1:  PR[91,1] = PR[90,1] + 34.527;
   1:  PR[91,2] = PR[90,2] + -19.507;
   1:  PR[91,3] = PR[90,3] + 50.154;
   1:L PR[91] R[100]mm/sec CNT100;
   1:  PR[91,1] = PR[90,1] + 35.214;
   1:  PR[91,2] = PR[90,2] + -18.985;
   1:  PR[91,3] = PR[90,3] + 50.169;
   1:L PR[91] R[100]mm/sec CNT100;
   1:  PR[91,1] = PR[90,1] + 35.683;
   1:  PR[91,2] = PR[90,2] + -18.727;
   1:  PR[91,3] = PR[90,3] + 50.172;
   1:L PR[91] R[100]mm/sec CNT100;
   1:  PR[91,1] = PR[90,1] + 36.774;
   1:  PR[91,2] = PR[90,2] + -17.985;
   1:  PR[91,3] = PR[90,3] + 50.173;
   1:L PR[91] R[100]mm/sec CNT100;
   1:  PR[91,1] = PR[90,1] + 39.923;
   1:  PR[91,2] = PR[90,2] + -19.381;
   1:  PR[91,3] = PR[90,3] + 50.177;
   1:L PR[91] R[100]mm/sec CNT100;
   1:  PR[91,1] = PR[90,1] + 41.587;
   1:  PR[91,2] = PR[90,2] + -20.216;
   1:  PR[91,3] = PR[90,3] + 50.188;
   1:L PR[91] R[100]mm/sec CNT100;
   1:  PR[91,1] = PR[90,1] + 43.821;
   1:  PR[91,2] = PR[90,2] + -21.034;
   1:  PR[91,3] = PR[90,3] + 50.194;
   1:L PR[91] R[100]mm/sec CNT100;
   1:  PR[91,1] = PR[90,1] + 46.682;
   1:  PR[91,2] = PR[90,2] + -21.974;
   1:  PR[91,3] = PR[90,3] + 50.201;
   1:L PR[91] R[100]mm/sec CNT100;
   1:  PR[91,1] = PR[90,1] + 49.780;
   1:  PR[91,2] = PR[90,2] + -22.524;
   1:  PR[91,3] = PR[90,3] + 50.210;
   1:L PR[91] R[100]mm/sec CNT100;
   1:  PR[91,1] = PR[90,1] + 52.452;
   1:  PR[91,2] = PR[90,2] + -23.068;
   1:  PR[91,3] = PR[90,3] + 50.220;
   1:L PR[91] R[100]mm/sec CNT100;
   1:  PR[91,1] = PR[90,1] + 53.948;
   1:  PR[91,2] = PR[90,2] + -23.338;
   1:  PR[91,3] = PR[90,3] + 50.228;
   1:L PR[91] R[100]mm/sec CNT100;
   1:  PR[91,1] = PR[90,1] + 56.988;
   1:  PR[91,2] = PR[90,2] + -23.393;
   1:  PR[91,3] = PR[90,3] + 50.233;
   1:L PR[91] R[100]mm/sec CNT100;
   1:  PR[91,1] = PR[90,1] + 61.230;
   1:  PR[91,2] = PR[90,2] + -23.399;
   1:  PR[91,3] = PR[90,3] + 50.242;
   1:L PR[91] R[100]mm/sec CNT100;
   1:  PR[91,1] = PR[90,1] + 66.789;
   1:  PR[91,2] = PR[90,2] + -22.440;
   1:  PR[91,3] = PR[90,3] + 50.255;
   1:L PR[91] R[100]mm/sec CNT100;
   1:  PR[91,1] = PR[90,1] + 68.521;
   1:  PR[91,2] = PR[90,2] + -21.919;
   1:  PR[91,3] = PR[90,3] + 50.273;
   1:L PR[91] R[100]mm/sec CNT100;
   1:  PR[91,1] = PR[90,1] + 71.740;
   1:  PR[91,2] = PR[90,2] + -20.701;
   1:  PR[91,3] = PR[90,3] + 50.278;
   1:L PR[91] R[100]mm/sec CNT100;
   1:  PR[91,1] = PR[90,1] + 75.153;
   1:  PR[91,2] = PR[90,2] + -18.845;
   1:  PR[91,3] = PR[90,3] + 50.289;
   1:L PR[91] R[100]mm/sec CNT100;
   1:  PR[91,1] = PR[90,1] + 76.365;
   1:  PR[91,2] = PR[90,2] + -18.088;
   1:  PR[91,3] = PR[90,3] + 50.301;
   1:L PR[91] R[100]mm/sec CNT100;
   1:  PR[91,1] = PR[90,1] + 80.368;
   1:  PR[91,2] = PR[90,2] + -14.622;
   1:  PR[91,3] = PR[90,3] + 50.305;
   1:L PR[91] R[100]mm/sec CNT100;
   1:  PR[91,1] = PR[90,1] + 80.906;
   1:  PR[91,2] = PR[90,2] + -13.881;
   1:  PR[91,3] = PR[90,3] + 50.321;
   1:L PR[91] R[100]mm/sec CNT100;
   1:  PR[91,1] = PR[90,1] + 83.228;
   1:  PR[91,2] = PR[90,2] + -10.553;
   1:  PR[91,3] = PR[90,3] + 50.324;
   1:L PR[91] R[100]mm/sec CNT100;
   1:  PR[91,1] = PR[90,1] + 83.372;
   1:  PR[91,2] = PR[90,2] + -10.330;
   1:  PR[91,3] = PR[90,3] + 50.337;
   1:L PR[91] R[100]mm/sec CNT100;
   1:  PR[91,1] = PR[90,1] + 84.966;
   1:  PR[91,2] = PR[90,2] + -6.208;
   1:  PR[91,3] = PR[90,3] + 50.338;
   1:L PR[91] R[100]mm/sec CNT100;
   1:  PR[91,1] = PR[90,1] + 85.181;
   1:  PR[91,2] = PR[90,2] + -5.613;
   1:  PR[91,3] = PR[90,3] + 50.351;
   1:L PR[91] R[100]mm/sec CNT100;
   1:  PR[91,1] = PR[90,1] + 85.792;
   1:  PR[91,2] = PR[90,2] + -0.729;
   1:  PR[91,3] = PR[90,3] + 50.353;
   1:L PR[91] R[100]mm/sec CNT100;
   1:  PR[91,1] = PR[90,1] + 85.181;
   1:  PR[91,2] = PR[90,2] + 4.154;
   1:  PR[91,3] = PR[90,3] + 50.368;
   1:L PR[91] R[100]mm/sec CNT100;
   1:  PR[91,1] = PR[90,1] + 84.965;
   1:  PR[91,2] = PR[90,2] + 4.749;
   1:  PR[91,3] = PR[90,3] + 50.383;
   1:L PR[91] R[100]mm/sec CNT100;
   1:  PR[91,1] = PR[90,1] + 83.372;
   1:  PR[91,2] = PR[90,2] + 8.871;
   1:  PR[91,3] = PR[90,3] + 50.385;
   1:L PR[91] R[100]mm/sec CNT100;
   1:  PR[91,1] = PR[90,1] + 83.228;
   1:  PR[91,2] = PR[90,2] + 9.094;
   1:  PR[91,3] = PR[90,3] + 50.399;
   1:L PR[91] R[100]mm/sec CNT100;
   1:  PR[91,1] = PR[90,1] + 80.906;
   1:  PR[91,2] = PR[90,2] + 12.423;
   1:  PR[91,3] = PR[90,3] + 50.400;
   1:L PR[91] R[100]mm/sec CNT100;
   1:  PR[91,1] = PR[90,1] + 80.369;
   1:  PR[91,2] = PR[90,2] + 13.163;
   1:  PR[91,3] = PR[90,3] + 50.412;
   1:L PR[91] R[100]mm/sec CNT100;
   1:  PR[91,1] = PR[90,1] + 76.360;
   1:  PR[91,2] = PR[90,2] + 16.632;
   1:  PR[91,3] = PR[90,3] + 50.415;
   1:L PR[91] R[100]mm/sec CNT100;
   1:  PR[91,1] = PR[90,1] + 75.139;
   1:  PR[91,2] = PR[90,2] + 17.394;
   1:  PR[91,3] = PR[90,3] + 50.431;
   1:L PR[91] R[100]mm/sec CNT100;
   1:  PR[91,1] = PR[90,1] + 71.723;
   1:  PR[91,2] = PR[90,2] + 19.251;
   1:  PR[91,3] = PR[90,3] + 50.436;
   1:L PR[91] R[100]mm/sec CNT100;
   1:  PR[91,1] = PR[90,1] + 68.474;
   1:  PR[91,2] = PR[90,2] + 20.474;
   1:  PR[91,3] = PR[90,3] + 50.448;
   1:L PR[91] R[100]mm/sec CNT100;
   1:  PR[91,1] = PR[90,1] + 66.752;
   1:  PR[91,2] = PR[90,2] + 20.991;
   1:  PR[91,3] = PR[90,3] + 50.458;
   1:L PR[91] R[100]mm/sec CNT100;
